           #tonSetStableWeight[#i](IN := #runTaimerStableWeight[#i],
                                   PT := t#250ms);

       ELSE
           #currentWeight[#i] := 0;
           #prevWeight[#i]:= 0;
       END_IF;

       IF #tonSetStableWeight[#i].Q OR #RS_TRIG_openBunker[#i] THEN
           IF #currentWeight[#i] <> "signalKVSStation".stableWeight[#i].weight[0] THEN
               "pushToArray"(addValue := #currentWeight[#i],
                             "array" := #stableWeight[#i].weight);
           END_IF;
           #runTaimerStableWeight[#i] := false;
       END_IF;


   END_FOR;
END_REGION
END_FUNCTION_BLOCK

FUNCTION_BLOCK "Sorting_AM"   // FB13, LAD
TITLE = Блок сортировки
{ S7_Optimized_Access := 'TRUE' }
VERSION : 0.1
// Из массива ReadyToSort считываем количество заполненых бункеров. Если их больше либо равно 6 то начинаем сортировку.
// После нахождения искомых бункеров формируем массив readyToDrop.
// После путем перемножения ReadyToSort *Not(readyToDrop) исключаем сбрасывемые бункера из сортировки
// stored: AutoNumber true, IsIECCheckEnabled false, IsRetainMemResEnabled false, MemoryReserve 100, SetENOAutomatically false, UDAEnableTagReadback false
   VAR_INPUT
      enableToWork : Bool;   // разрешение на работу блока
      setWeight : Real;   // итоговый разыскиваемый вес
      errorMeasurement : Real;   // погрешность
      isWorkWithBunker : Array[0..12] of Bool;   // разрешение работать с конкретными бункерами
      setWeightBunker { ExternalAccessible := 'False'; ExternalVisible := 'False'; ExternalWritable := 'False'} : Array[0..12] of Real;   // уставки весов в бункерах
   END_VAR
   VAR_IN_OUT
      stableWeightBunker : Array[0..12] of Real;   // стабильный вес в бункерах
      readyToSorting : Array[0..12] of Bool;   // готовность бункеров к сортировке
      readyToDrop : Array[0..12] of Bool;   // итоговый сигнал сортировки для сброса на конвейер
      blockSort : Bool;   // блокировать сортировку чтобы просто скинуть все готовые
   END_VAR
   VAR
      valueReadyToDrop { ExternalAccessible := 'False'; ExternalVisible := 'False'; ExternalWritable := 'False'} : Bool;
      valueReadytoSortBunker : SInt;   // количество бункеров готовых к сортировке
      valueIsWorkWithBunker : SInt;
      tmpStableWeight : Array[0..12] of Real;   // массив с весами которые будем сортировать
      bufferReadyToDrop : Array[0..12] of Bool;   // на случай того что если readyToDrop не был сброшен
      Sort_Real_FB : "Sort_Real";
      full1 : Array[0..12] of Bool;
      full0 : Array[0..12] of Bool;
      pow2_DB : "pow2";
      minValue : Real;
      minValueArray : Array[0..12] of Bool;
      tmpArrNotDrop { ExternalAccessible := 'False'; ExternalVisible := 'False'; ExternalWritable := 'False'} : Array[0..12] of Real;
      tmpSumFind { ExternalAccessible := 'False'; ExternalVisible := 'False'; ExternalWritable := 'False'} : Real;
      valueMaxSortFor { ExternalAccessible := 'False'; ExternalVisible := 'False'; ExternalWritable := 'False'} : Int;   // максимальное число циклов для нахождения искомого веса
      bitMaskSortFor { ExternalAccessible := 'False'; ExternalVisible := 'False'; ExternalWritable := 'False'} : Array[0..12] of Bool;
      stateFindIndex { ExternalAccessible := 'False'; ExternalVisible := 'False'; ExternalWritable := 'False'} : Bool;
      tmpReadyToDrop { ExternalAccessible := 'False'; ExternalVisible := 'False'; ExternalWritable := 'False'} : Array[0..12] of Bool;   // временный массив готовности к сбросу
      tabActiveSort { ExternalAccessible := 'False'; ExternalVisible := 'False'; ExternalWritable := 'False'} : Bool;
      saveBitMaskSortFor { ExternalAccessible := 'False'; ExternalVisible := 'False'; ExternalWritable := 'False'} : Array[0..12] of Bool;
   END_VAR
   VAR_TEMP
      i : DInt;
      j : DInt;
      k : DInt;
      l : DInt;
      "m" : DInt;
      it : DInt;
      one : DInt;
      indexTmpSumFind : DInt;
      valueOneBitMask : DInt;
   END_VAR
   // full1[1..12] := true;
BEGIN

REGION Network 1 (SCL): Определяем ValueToSortBunker
   #tmpReadyToDrop := #full0;
   IF #enableToWork THEN //разрешение на работу блока 
       //необходимо проверить не подготовил ли блок сортировки уже значения для сброса
       #valueReadyToDrop := false;
       #i := 0;
       FOR #i := 1 TO 12 DO
           IF #readyToDrop[#i] THEN
               #valueReadyToDrop := true;
               EXIT;//выходим из FOR тк то что надо уже нашли
           END_IF;
       END_FOR;

       IF NOT (#valueReadyToDrop) THEN
           //если сортировку не производили
           #i := 0;
           #valueIsWorkWithBunker := 0;
           #valueReadytoSortBunker := 0;
           FOR #i := 1 TO 12 DO
               //подсчитаем количесво бункеров с которыми можно работать
               //и какие готовы к сортировке
               //
               IF #isWorkWithBunker[#i] THEN
                   #valueIsWorkWithBunker := #valueIsWorkWithBunker + 1;
               END_IF;
               IF #readyToSorting[#i] AND #isWorkWithBunker[#i] THEN
                   #valueReadytoSortBunker := #valueReadytoSortBunker + 1;
               END_IF;
           END_FOR;

           IF #blockSort THEN
               //если включена блокировка то просто ждем готовности бункеров к сортировке
               //
               IF #valueIsWorkWithBunker = #valueReadytoSortBunker THEN
                   //если число готовых к сортировке бункеров совпадает 
                   //с числом разрешенных к работе в режиме блокировки то
                   //просто скидываем все
                   #tmpReadyToDrop := #readyToSorting;
               END_IF;
           ELSE
               //если блокировки нет то сортируем по стандарту

               // IF #valueIsWorkWithBunker = 1 THEN
               //     //если бункеров разрешенных к работе один то 
               //     #i := 0;
               //     FOR #i := 1 TO 12 DO //заполняем временный массив готовности к сбросу
               //         #tmpReadyToDrop[#i] := #readyToSorting[#i] AND #isWorkWithBunker[#i];
               //     END_FOR;
               // ELSE

               //IF #valueReadytoSortBunker >= 3 THEN//начинаем сортировку
               IF #valueReadytoSortBunker =12 THEN//начинаем сортировку
                   #i := 0;
                   FOR #i := 1 TO 12 DO//определим массив чисел с которыми будем работать
                       #tmpStableWeight[#i] := #stableWeightBunker[#i] * BOOL_TO_INT(#readyToSorting[#i]);
                   END_FOR;
                   //далее работаем только с весами из массива #tmpStableWeight
                   //
                   REGION
                       // // //*****************************
                       // // //временная заглушка - скидываем бункера которые тупа в сумме
                       // // //дают больше либо равно уставке
                       // // //
                       // #tmpArrNotDrop := #tmpStableWeight;


                       // //#Sort_Real_FB(array := #tmpArrNotDrop,sortDirection:=true);
                       // //теперь массив #tmpArrNotDrop отсортирован и числа которые 
                       // //мы можем использовать начинаются с индекса (12-noDrop+1)
                       // #k := 0;
                       // #tmpSumFind := 0;//где храним сумму
                       // #stateFindIndex := false;
                       // #indexTmpSumFind := 0;//индекс элемента массива на котором надо остановиться
                       // //#noDrop := #valueReadytoSortBunker;
                       // FOR #k := 0 TO 12 DO
                       //     #tmpSumFind := #tmpSumFind + #tmpArrNotDrop[#k];
                       //     IF #tmpSumFind >= #setWeight//если попадаем 
                       //     THEN
                       //         #stateFindIndex := true;
                       //         #indexTmpSumFind := #k;
                       //         EXIT;//выходим из FOR
                       //     END_IF;

                       // END_FOR;
                       // IF NOT (#stateFindIndex) THEN //ничего не нашли
                       //     #tmpReadyToDrop := #full0;
                       // ELSE
                       //     #l := 0;//заполняем массив на сброс
                       //     FOR #l := 1 TO #indexTmpSumFind DO
                       //         IF #tmpArrNotDrop[#l] > 0 THEN
                       //             #tmpReadyToDrop[#l] := true;
                       //         ELSE
                       //             #tmpReadyToDrop[#l] := false;
                       //         END_IF;
                       //     END_FOR;

                       // END_IF;
                       // // // //*************************************
                   END_REGION ;
                   REGION
                       //****************
                       //сортировка на основе двоичного представления числа
                       //
                       #tmpArrNotDrop := #tmpStableWeight;
                       #Sort_Real_FB("array" := #tmpArrNotDrop,
                                     sortDirection := true);
                       // //теперь массив #tmpArrNotDrop отсортирован в порядке убывания и 
                       //только необходимо обратить внимание что все веса начинаются с 0 индекса
                       #pow2_DB(basic := #valueReadytoSortBunker,
                                pow := #valueMaxSortFor);
                       #it := 0;
                       #stateFindIndex := false;
                       #minValue := 99999;
                       #minValueArray := #full0;
                       #tabActiveSort := false;
                       FOR #it := 1 TO #valueMaxSortFor DO
                           // // #bitMaskSortFor[0] := #it.%X0;
                           // // #bitMaskSortFor[1] := #it.%X1;
                           // // #bitMaskSortFor[2] := #it.%X2;
                           // // #bitMaskSortFor[3] := #it.%X3;
                           // // #bitMaskSortFor[4] := #it.%X4;
                           // // #bitMaskSortFor[5] := #it.%X5;
                           // // #bitMaskSortFor[6] := #it.%X6;
                           // // #bitMaskSortFor[7] := #it.%X7;
                           // // #bitMaskSortFor[8] := #it.%X8;
                           // // #bitMaskSortFor[9] := #it.%X9;
                           // // #bitMaskSortFor[10] := #it.%X10;
                           // // #bitMaskSortFor[11] := #it.%X11;
                           // // #bitMaskSortFor[12] := #it.%X12;
                           // // #tmpSumFind := #tmpArrNotDrop[0] * BOOL_TO_SINT(#bitMaskSortFor[0]) +
                           // // #tmpArrNotDrop[1] * BOOL_TO_SINT(#bitMaskSortFor[1]) +
                           // // #tmpArrNotDrop[2] * BOOL_TO_SINT(#bitMaskSortFor[2]) +
                           // // #tmpArrNotDrop[3] * BOOL_TO_SINT(#bitMaskSortFor[3]) +
                           // // #tmpArrNotDrop[4] * BOOL_TO_SINT(#bitMaskSortFor[4]) +
                           // // #tmpArrNotDrop[5] * BOOL_TO_SINT(#bitMaskSortFor[5]) +
                           // // #tmpArrNotDrop[6] * BOOL_TO_SINT(#bitMaskSortFor[6]) +
                           // // #tmpArrNotDrop[7] * BOOL_TO_SINT(#bitMaskSortFor[7]) +
                           // // #tmpArrNotDrop[8] * BOOL_TO_SINT(#bitMaskSortFor[8]) +
                           // // #tmpArrNotDrop[9] * BOOL_TO_SINT(#bitMaskSortFor[9]) +
                           // // #tmpArrNotDrop[10] * BOOL_TO_SINT(#bitMaskSortFor[10]) +
                           // // #tmpArrNotDrop[11] * BOOL_TO_SINT(#bitMaskSortFor[11]) +
                           // // #tmpArrNotDrop[12] * BOOL_TO_SINT(#bitMaskSortFor[12]);
                           // 
                           #tmpSumFind :=
                           #tmpArrNotDrop[0] * BOOL_TO_SINT(#it.%X0) +
                           #tmpArrNotDrop[1] * BOOL_TO_SINT(#it.%X1) +
                           #tmpArrNotDrop[2] * BOOL_TO_SINT(#it.%X2) +
                           #tmpArrNotDrop[3] * BOOL_TO_SINT(#it.%X3) +
                           #tmpArrNotDrop[4] * BOOL_TO_SINT(#it.%X4) +
                           #tmpArrNotDrop[5] * BOOL_TO_SINT(#it.%X5) +
                           #tmpArrNotDrop[6] * BOOL_TO_SINT(#it.%X6) +
                           #tmpArrNotDrop[7] * BOOL_TO_SINT(#it.%X7) +
                           #tmpArrNotDrop[8] * BOOL_TO_SINT(#it.%X8) +
                           #tmpArrNotDrop[9] * BOOL_TO_SINT(#it.%X9) +
                           #tmpArrNotDrop[10] * BOOL_TO_SINT(#it.%X10) +
                           #tmpArrNotDrop[11] * BOOL_TO_SINT(#it.%X11);

                           IF #tmpSumFind >= #setWeight AND #tmpSumFind <= (#setWeight + (#setWeight * #errorMeasurement / 100))
                           THEN
                               #stateFindIndex := true;
                               EXIT;
                               ;
                           ELSE
                               IF (#tmpSumFind > #setWeight) AND (#tmpSumFind < #minValue) THEN
                                   #minValue := #tmpSumFind;
                                   "bitMaskSortFor"(value := #it,
                                                    bitMask := #bitMaskSortFor);
                                   #minValueArray := #bitMaskSortFor;
                               END_IF;
                           END_IF;


                       END_FOR;
                       //на выходе мы имеем битовую маску которая лучше всего подходит
                       //
                       //также обрабатываем условие что карманы все заняты а чтото скинуть надо
                       IF NOT (#stateFindIndex) THEN //
                           IF #valueReadytoSortBunker > 10 THEN
                               #tabActiveSort := TRUE;
                               #saveBitMaskSortFor := #minValueArray;
                           END_IF;
                       ELSE
                           #tabActiveSort := true;
                           "bitMaskSortFor"(value := #it,
                                            bitMask := #bitMaskSortFor);
                           #saveBitMaskSortFor := #bitMaskSortFor;
                       END_IF;
                       #tmpReadyToDrop := #full0;
                       //определяем финальный tmpReadyToDrop
                       IF #tabActiveSort THEN
                           //если активированная нахождение искомых бункеров
                           #l := 0;
                           FOR #l := 0 TO 12 DO
                               IF #saveBitMaskSortFor[#l] AND ((BOOL_TO_INT(#saveBitMaskSortFor[#l]) * #tmpArrNotDrop[#l]) > 0) THEN
                                   #k := 0;
                                   FOR #k := 1 TO 12 DO
                                       IF #tmpArrNotDrop[#l] = #tmpStableWeight[#k] THEN
                                           #tmpReadyToDrop[#k] := true;
                                           EXIT;
                                       END_IF;
                                   END_FOR;
                               END_IF;
                           END_FOR;
                       END_IF;
                   END_REGION
                   //корректируем массив readyToSorting
                   #i := 0;
                   FOR #i := 1 TO 12 DO
                       IF #tmpReadyToDrop[#i] THEN
                           #readyToSorting[#i] := false;
                       END_IF;
                   END_FOR;
               END_IF;
           END_IF;
       ELSE
           #tmpReadyToDrop := #readyToDrop;//если значения уже были
           //и не сброшены то сортировку не производили
       END_IF;

   END_IF;



   #readyToDrop := #tmpReadyToDrop;//переписываем из временного в блочный
END_REGION
END_FUNCTION_BLOCK

FUNCTION_BLOCK "pow2"
{ S7_Optimized_Access := 'TRUE' }
VERSION : 0.1
   VAR_INPUT 
      basic : SInt;   // степень возведение двойки
   END_VAR

   VAR_IN_OUT 
      pow : Int;   // ответ возведения -1
   END_VAR


BEGIN
	CASE #basic OF //
	    1:
	       #pow:=1;
	    2:  
	        #pow:=3;
	    3:
	        #pow:=7;
	    4:
	        #pow:=15;
	    5:
	        #pow:=31;
	    6:
	        #pow:=63;
	    7:
	        #pow:=127;
	    8:
	        #pow:=255;
	    9:
	        #pow:=511;
	    10:
	        #pow:=1023;
	    11:
	        #pow:=2047;
	    12:
	        #pow:=4095;
	END_CASE;
	
END_FUNCTION_BLOCK

FUNCTION_BLOCK "setWeightBunker_AM"   // FB3, LAD
{ S7_Optimized_Access := 'TRUE' }
VERSION : 0.1
// Блок уставок, работы упаковочных машин.
// Определяет уставки для бункеров. Дают разрешение на работу бункера.
// Даже если сброшено меньше 
// Говорит о готовности упаковочных машин принять дозу и в какую машину скидывать
// stored: AutoNumber true, IsIECCheckEnabled false, IsRetainMemResEnabled false, MemoryReserve 100, SetENOAutomatically false, UDAEnableTagReadback false
   VAR_INPUT
      enableWork : Bool;   // разрешение работы блока
      weightPack : Real;   // заданный вес упаковки
      measurementError : Real;   // погрешность
      maxWeightBunker : Real;   // максимальный вес в бункере
      mediumWeightProduct : Real;   // средний вес продукта
   END_VAR
   VAR_IN_OUT
      taskWeightBunker : Real;   // целевой вес который ищем в сортировке
      setWeightBunker : Array[0..12] of Real;   // уставки задаваемые в бункера
      isWorkWithBunker : Array[0..12] of Bool;   // разрешение работать с конкретными бункерами
      readyToDrop : Array[0..12] of Bool;   // массив который будет сбрасываться
      YP_ReadyToDrop : Array[0..2] of Bool;   // сигнал говорит о том что в УМ можно 100% чтото скинуть
      stableWeightBunker : Array[0..12] of Real;   // стабильный вес в бункерах
      blockSort : Bool;   // запрещение работы сортировки в блоке сортировки
   END_VAR
   VAR
      measureErrorGramm : Real;   // погрешность измерения в граммах
      dropWeight : Real;   // уже сброшенный вес
      hmiDropWeight : Real;   // отображаемый сброшенный вес на панеле
      hmiMeasurementError : Real;   // отображаемая сброшенная погрешность на панеле
      indexLastDropYP : SInt;   // индекс машины в которую последний раз сбрасывали
      full1 : Array[0..12] of Bool;
      full0 : Array[0..12] of Bool;
      Sort_Real_FB : "Sort_Real";
   END_VAR
   VAR_TEMP
      i : DInt;
      j : DInt;
      k : DInt;
      l : DInt;
      "m" : DInt;
      expX : Real;
      expY : Real;
      tmpNeedWeight : Real;
      tmpc1 : Real;
      tmpc2 : DInt;
      tmpc3 : Real;
      minSearch : Real;   // минимальное найденое число остаточном массиве
      indexMinSearch : DInt;   // индекс минимального числа
      isSearchSuccess : Bool;   // поиск прошел успешно
      indexSearchSuccess : DInt;   // индекс оставшегося идеального кармана
      valueDropBunker : DInt;
      tmpArrNotDrop : Array[0..12] of Real;
      tmpArrWeightNoDrop : Array[0..12] of Real;
      noDrop : Int;
      tmpSumFind : Real;
      indexTmpSumFind : DInt;
   END_VAR
   // full1[1..12] := true;
BEGIN

REGION Network 1 (SCL): переведем погрешность в граммы
   #measureErrorGramm := #measurementError * #weightPack / 100;
END_REGION

REGION Network 2 (SCL): Определяем уставки в карманы и выставляем разрешения работы
   // на основе веса который мы уже сбросили и который будем сбрасывать 
   // а также учитывая веса в рецепте определяем уставки в карманах, целевую уставку для поиска, а также 
   // выставляем разрешения работы по конкретным бункерам
   IF #enableWork THEN

       //*********************************************
       //определение сброшенного веса на основе массивов со стабильными весами
       //и массива ячеек которые должны быть сброшены. Обнуление сброшенного веса в случае 
       //выполнения условия
       //также производим этот расчет только при условии что мы сбросим кудато этот вес
       IF #YP_ReadyToDrop[1] OR #YP_ReadyToDrop[2] THEN
           #i := 0;
           FOR #i := 1 TO 12 DO
               #dropWeight := #dropWeight + BOOL_TO_INT(#readyToDrop[#i]) * #stableWeightBunker[#i];
           END_FOR;
           // #hmiDropWeight := #dropWeight;
           // #hmiMeasurementError := (#weightPack - #dropWeight) / #weightPack;
           IF #dropWeight >= #weightPack THEN
               #dropWeight := 0;
           END_IF;
       END_IF;
       //************************************


       //основное распространение весов, когда выкидываем весь вес за раз
       //

       #expX := #weightPack / 10;//#weightPack / 6;
       #expY := #mediumWeightProduct / 3;

       //если #expX<=MAX_WEIGHT_BUNKER то работаем по стандарту,
       //иначе ограничеваем #expX=MAX_WEIGHT_BUNKER
       IF #expX > #maxWeightBunker THEN
           #expX := #maxWeightBunker;
       END_IF;

       IF #dropWeight = 0 THEN
           // #j := 2;
           // WHILE (6 * #expX) < #weightPack + #j * #expY AND #j <> 0 DO
           //     #j := #j - 1;
           // END_WHILE;
           // #expY := (#expY / 2) * #j;//корректировка #expY
           #taskWeightBunker := #weightPack;//вес для поиска по рецепту
           #isWorkWithBunker := #full1;//разрешаем работу всем линиям

           #setWeightBunker[1] := #setWeightBunker[6] :=
           #setWeightBunker[7] := #setWeightBunker[12] := #expX;

           #setWeightBunker[2] := #setWeightBunker[5] :=
           #setWeightBunker[8] := #setWeightBunker[11] := #expX - #expY;

           #setWeightBunker[3] := #setWeightBunker[4] :=
           #setWeightBunker[9] := #setWeightBunker[10] := #expX - 2 * #expY;

       ELSE//если уже сбрасываем

           #valueDropBunker := 0;//определяем сбрасываем ли мы чтото чтобы запретить
           //перерасчет в этом условии
           //просто на первой итерации как только сюда поступает массив readyToDrop
           //мы выставляем требуемые уставки, а потом запрещаем их изменять
           #k := 0;
           FOR #k := 1 TO 12 DO
               #valueDropBunker := #valueDropBunker + BOOL_TO_SINT(#readyToDrop[#k]);
           END_FOR;

           IF #valueDropBunker > 0 THEN
               //следующий просчет актуален только на итерации перед сбросом веса поэтому 
               //после сброса на конвейер эту часть надо блокировать для изменений
               //
               //только еще надо обыгрывать момент когда сбрасываются сразу 12 бункеров

               #tmpNeedWeight := #weightPack - #dropWeight;//вес остатка

               IF #valueDropBunker < 12 THEN //при сбрасывании всех 12 бункеров
                   //будет другой механизм выдачи разрешений

                   IF #tmpNeedWeight <= #expX THEN //если нужно докинуть меньше чем в одном бункере,то
                       //ищем вес совпадающий с остатком и если такой не находим
                       //то берем минимальную ячейку с весом

                       #minSearch := 99999.9;//берется как минимальное тк такое точно не будет в бункере
                       #k := 0;
                       #isSearchSuccess := false;
                       FOR #k := 1 TO 12 DO//ищем бункер идеально подходящий по весу и параллельно ведем
                           //поиск первого минимального числа

                           IF NOT (#readyToDrop[#k]) THEN
                               IF #stableWeightBunker[#k] < #minSearch THEN
                                   //параллельно ищем минимальное число
                                   #minSearch := #stableWeightBunker[#k];
                                   #indexMinSearch := #k;
                               END_IF;

                               IF (#tmpNeedWeight <= #stableWeightBunker[#k]//проверяем оставшиеся карманы на вес
                                   AND #stableWeightBunker[#k] <= #tmpNeedWeight + #measureErrorGramm / 6) THEN
                                   #isSearchSuccess := true;
                                   #indexSearchSuccess := #k;//сохраняем индекс идеального кармана
                                   EXIT;//выходим из FOR
                               END_IF;
                           END_IF;

                       END_FOR;
                       //если идеальный карман так и не найдем 
                       //берем карман с минимальным весом и перемещаем его индекс в #indexSearchSuccess
                       IF NOT (#isSearchSuccess) THEN
                           #indexSearchSuccess := #indexMinSearch;
                       END_IF;

                       #taskWeightBunker := #tmpNeedWeight;//вес для поиска в сортировке
                       #isWorkWithBunker := #full0;//запрещаем работу всем линиям
                       #isWorkWithBunker[#indexSearchSuccess] := true;//включаем только нужную линию
                       #setWeightBunker[#indexSearchSuccess] := #tmpNeedWeight;
                       #blockSort := true;//выставляем блокировку тк надо будет только сбросить

                   ELSE//если докидывать больше чем в одном бункере
                       #k := 0;//выделяем веса которые не сбрасываются
                       FOR #k := 1 TO 12 DO
                           IF NOT (#readyToDrop[#k]) THEN
                               #noDrop := #noDrop + 1;//колво добавленных элементов
                               #tmpArrNotDrop[#k] := #stableWeightBunker[#k];
                           END_IF;
                       END_FOR;
                       //будем использовать #tmpArrWeightNoDrop для поиска искомых бункеров
                       #tmpArrWeightNoDrop := #tmpArrNotDrop;

                       #Sort_Real_FB("array" := #tmpArrNotDrop);
                       //теперь массив #tmpArrNotDrop отсортирован и числа которые 
                       //мы можем использовать начинаются с индекса (12-noDrop+1)
                       #k := 0;
                       #tmpSumFind := 0;//где храним сумму
                       #indexTmpSumFind := 0;//индекс элемента массива на котором надо остановиться
                       FOR #k := (12 - #noDrop + 1) TO 12 DO
                           #tmpSumFind := #tmpSumFind + #tmpArrNotDrop[#k];
                           IF #tmpSumFind >= #tmpNeedWeight//если попадаем идеально
                               AND #tmpSumFind <= #tmpNeedWeight + #measureErrorGramm THEN
                               #indexTmpSumFind := #k;
                               EXIT;//выходим из FOR
                           END_IF;
                           //если превысили сумму
                           IF #tmpSumFind > #tmpNeedWeight + #measureErrorGramm THEN
                               #indexTmpSumFind := #k - 1;
                               EXIT;
                           END_IF;
                           IF #k = 12 THEN
                               #indexTmpSumFind := #k;
                           END_IF;
                       END_FOR;
                       //теперь проверим чтобы #indexTmpSumFind входил в массив с весами
                       //потому что первый же вес может быть больше того что мы исчем
                       IF #tmpArrNotDrop[#indexTmpSumFind] <> 0 THEN
                           #taskWeightBunker := #tmpNeedWeight;//вес для поиска по рецепту
                           #isWorkWithBunker := #full0;//запрещаем работу всем линиям
                           #blockSort := true;//выставляем блокировку тк надо будет только
                           //дождать сигналов готовности к сортировке сбросить

                           //теперь заполняем массив разрешения работ через поиск весов
                           //и параллельно выставляем уставки
                           IF #tmpSumFind >= #tmpNeedWeight//если попадаем идеально
                               AND #tmpSumFind <= #tmpNeedWeight + #measureErrorGramm THEN
                               //если вес сходился 
                               #l := 0;
                               FOR #l := (12 - #noDrop + 1) TO #indexTmpSumFind DO
                                   #m := 0;
                                   FOR #m := 1 TO 12 DO//ищем отсортированные веса и сопоставляем их индексы
                                       //ищем в заранее сохранненом массивве с весам который не сбрасываются
                                       //и имеют правильные индексы
                                       IF #tmpArrWeightNoDrop[#m] = #tmpArrNotDrop[#l] THEN
                                           #isWorkWithBunker[#m] := true;
                                           #setWeightBunker[#m] := #tmpArrWeightNoDrop[#m];
                                           EXIT;//ищем следующий вес
                                       END_IF;
                                   END_FOR;
                               END_FOR;

                           ELSE //сюда поподем если веса с излишкой или недостаточно 
                               //если вес не сходился
                               #l := 0;
                               FOR #l := (12 - #noDrop + 1) TO #indexTmpSumFind DO
                                   #m := 0;
                                   FOR #m := 1 TO 12 DO
                                       IF #tmpArrWeightNoDrop[#m] = #tmpArrNotDrop[#l] THEN
                                           #isWorkWithBunker[#m] := true;
                                           #setWeightBunker[#m] := #tmpNeedWeight / DINT_TO_INT((#indexTmpSumFind - (12 - #noDrop + 1)));
                                           EXIT;//ищем следующий вес
                                       END_IF;
                                   END_FOR;
                               END_FOR;


                           END_IF;
                           ;

                       END_IF;

                   END_IF;
               ELSE //а теперь что делать если сброшены все 12
                   //надо вводить какойто новый сигнал который сказал бы нагружать бункера только после закрытия? или 
                   //все успеется
                   //!!!обратить внимание на это
                   //

                   //расчитываем сколько бункеров необходимо для сбора оставшегося веса
                   //это делаем на основе максимального веса в бункере
                   //
                   #taskWeightBunker := #tmpNeedWeight;//вес для поиска в сортировке
                   #blockSort := true;//выставляем блокировку тк надо будет только скинуть
                   #tmpc2 := ROUND(#tmpNeedWeight / #maxWeightBunker); //число используемых бункеров
                   #i := 0;
                   FOR #i := 1 TO #tmpc2 DO
                       #isWorkWithBunker[#k] := true;
                       #setWeightBunker[#k] := #tmpNeedWeight / DINT_TO_REAL(#tmpc2);
                   END_FOR;
                   ;
               END_IF;
           END_IF;
       END_IF;


   ELSE
       #isWorkWithBunker := #full0;//запрет на работу все бункерам
   END_IF;
END_REGION
END_FUNCTION_BLOCK

FUNCTION_BLOCK "workPackingMachine_AM"   // FB4, LAD
TITLE = Работа с УМ, бункерами
{ S7_Optimized_Access := 'TRUE' }
VERSION : 0.1
// stored: AutoNumber true, IsIECCheckEnabled false, IsRetainMemResEnabled false, MemoryReserve 100, SetENOAutomatically false, UDAEnableTagReadback false
   VAR_INPUT
      enWork : Bool;   // разрешение работы
      YP_ReadyAccept : Array[0..2] of Bool;   // сигнал от упак машины что готова принять
      YP_StartDozing : Array[0..2] of Bool;   // сигнал от упаковочной машины что начать дозирование
      weightPack : Real;   // заданный вес упаковки
   END_VAR
   VAR_IN_OUT
      hmiYpDropWeight : Array[0..2] of Real;   // вывод на панель сброшенного веса
      hmiYPDropErrorMeasure : Array[0..2] of Real;   // вывод на панель погрешности
      openLeftBunker : Array[0..12] of Bool;   // сгналы открытия левых бункеров
      closeLeftBunker : Array[0..12] of Bool;   // сигналы закрытия левых бункеров
      openRightBunker : Array[0..12] of Bool;   // сигналы открытия правых бункеров
      closeRightBunker : Array[0..12] of Bool;   // сигналы закрытия правых бункеров
      alarmStop : Bool;   // аварийный останов
      Yq_ReadyDoze : Array[0..2] of Bool;   // сигнал на упаковочную машину что доза готова
      YP_ReadyToDrop : Array[0..2] of Bool;   // сигнал говорит о том что в УМ можно 100% чтото скинуть
      stableWeightBunker : Array[0..12] of Real;   // стабильный вес в бункерах
      readyToSort : Array[0..12] of Bool;
      readyToDrop : Array[0..12] of Bool;   // массив который будет сбрасываться
      Conv_FRV : Array[0..2] of Bool;   // запуск конвейеров вперед
      Conv_REV : Array[0..2] of Bool;   // запуск конвейеров назад
   END_VAR
   VAR
      dropLeftBunker { ExternalAccessible := 'False'; ExternalVisible := 'False'; ExternalWritable := 'False'} : Array[0..12] of Bool;   // массив на сброс левых бункеров
      dropRightBunker { ExternalAccessible := 'False'; ExternalVisible := 'False'; ExternalWritable := 'False'} : Array[0..12] of Bool;   // массив на сброс правых бункеров
      tmpPtrig : Array[0..1] of Bool;
      dropTon : Array[0..2] of TON_TIME;   // выдержка на передачу сигнала УМ ДОЗА
      startDropTon : Array[0..2] of Bool;   // начало отсчета для таймера
      dropWeight : Real;   // сбрасываемый вес
      nextDropConveyer : SInt;   // индекс конвейера на который сбрасывали последним
      tonReadyDozeTimer : Array[0..2] of TON_TIME;
      leftBunker_FB : Array[0..12] of "controlValve";
      rightBunker_FB : Array[0..12] of "controlValve";
      full1 : Array[0..12] of Bool;
      full0 : Array[0..12] of Bool;
      valueDropBunker : Bool;
      watchDrop : Array[0..12] of Bool;
      F_TRIG_Instance { S7_SetPoint := 'True'} : F_TRIG;
   END_VAR
   VAR_TEMP
      i : DInt;
      resetTimerDropYp : Array[0..2] of Bool;
      resetTimerDropTon : Array[0..2] of Bool;
   END_VAR
   // full1[1..12] := true;
   VAR_TEMP   // added for the SCL form of the ladder/FBD networks
      _w1 : Bool;
      _w2 : Bool;
   END_VAR
BEGIN

REGION Network 1: сброс вращения если убрать сигнал разрешения
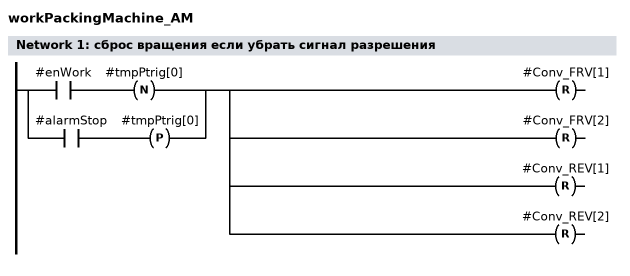
   RUNG wire#powerrail
      Contact( #enWork )
      N_Trig( #tmpPtrig[0] )
      wire#w1
      R_Coil( #Conv_FRV[1] )
   END_RUNG
   RUNG wire#powerrail
      Contact( #alarmStop )
      P_Trig( #tmpPtrig[0] )
   END_RUNG wire#w1
   RUNG wire#w1
      R_Coil( #Conv_FRV[2] )
   END_RUNG
   RUNG wire#w1
      R_Coil( #Conv_REV[1] )
   END_RUNG
   RUNG wire#w1
      R_Coil( #Conv_REV[2] )
   END_RUNG
   // the same network as SCL:
   #_w1 := NOT #enWork AND #tmpPtrig[0];   // falling edge
   #tmpPtrig[0] := #enWork;
   #_w2 := #alarmStop AND NOT #tmpPtrig[0];   // rising edge
   #tmpPtrig[0] := #alarmStop;
   IF #_w1 OR #_w2 THEN
       #Conv_FRV[1] := FALSE;
       #Conv_FRV[2] := FALSE;
       #Conv_REV[1] := FALSE;
       #Conv_REV[2] := FALSE;
   END_IF;
END_REGION

REGION Network 2 (SCL): Подсчет сбрасываемых бункеров
   #i := 0;
   #valueDropBunker := FALSE;
   FOR #i := 1 TO 12 DO
       IF #readyToDrop[#i] THEN
           #valueDropBunker := true;
           EXIT;
       END_IF;
   END_FOR;
END_REGION

REGION Network 3 (SCL): Сброс сигнала на УМ #Yq_ReadyDoze
   #i := 0;
   FOR #i := 1 TO 2 DO
       // IF #Yq_ReadyDoze[#i] THEN
       //     #Yq_ReadyDoze[#i] := false;
       // END_IF;
       #tonReadyDozeTimer[#i](IN := #Yq_ReadyDoze[#i],
                              PT := t#1s,
                              Q => #resetTimerDropYp[#i]);

   END_FOR;
   #i := 0;
   FOR #i := 1 TO 2 DO

       IF #resetTimerDropYp[#i] THEN
           #Yq_ReadyDoze[#i] := false;
       END_IF;

   END_FOR;
END_REGION

REGION Network 4 (SCL): Формирование сигналов
   // #YP_ReadyToDrop
   #i := 0;
   FOR #i := 1 TO 2 DO
       #YP_ReadyToDrop[#i] := #YP_ReadyAccept[#i] AND #YP_StartDozing[#i] AND NOT(#startDropTon[#i]) AND NOT(#Yq_ReadyDoze[#i]);
   END_FOR;
END_REGION

REGION Network 5 (SCL): учет сбрасываемого веса
   // помещаем в переменнную #dropWeight вес который будет сброшен
   IF #enWork THEN
       IF (#YP_ReadyToDrop[1] OR #YP_ReadyToDrop[2]) AND #valueDropBunker THEN
           #i := 0;
           FOR #i := 1 TO 12 DO
               #dropWeight := #dropWeight + BOOL_TO_INT(#readyToDrop[#i])
               * #stableWeightBunker[#i];
           END_FOR;
       END_IF;
   END_IF;
END_REGION

REGION Network 6 (SCL): вращение конвейеров
   //"hmi".outConvAndPack[1].isUseInBegin - разрешение использовать
   // "hmi".outConvAndPack[1].isUpInBegin - вращать вперед
   #i := 0;
   FOR #i := 1 TO 2 DO
       IF #enWork AND "hmi".outConvAndPack[#i].isUseInBegin THEN
           IF "hmi".outConvAndPack[#i].isUpInBegin THEN
               #Conv_FRV[#i] := true;
               #Conv_REV[#i] := false;
           ELSE
               #Conv_FRV[#i] := false;
               #Conv_REV[#i] := true;
           END_IF;
       ELSE
           #Conv_FRV[#i] := false;
           #Conv_REV[#i] := false;
       END_IF;
   END_FOR;
END_REGION

REGION Network 7 (SCL): Формирование сигнала доза готова
   IF #enWork THEN
       IF #valueDropBunker THEN//определяем какие бункеры открываем
           //, а также даем отсечку времени для отправки
           //ДОЗА ГОТОВА
           IF #YP_ReadyToDrop[1] OR #YP_ReadyToDrop[2] THEN
               //ПРОСТО ЕСЛИ НЕ СКИДЫВАЕМ ТО И НЕ НАДО ОЧИЩАТЬ МАССИВ READYTOdROP
               IF #YP_ReadyToDrop[1] AND #YP_ReadyToDrop[2] THEN
                   //если оба доступны то по следующему индексу
                   CASE #nextDropConveyer OF
                       0, 2:  //следующий был второй
                           IF #Conv_FRV[2] THEN
                               #hmiYpDropWeight[1] := #dropWeight;
                               #hmiYPDropErrorMeasure[1] := (#weightPack - #dropWeight) / #weightPack * 100;
                               #startDropTon[1] := true;
                           ELSE
                               #hmiYpDropWeight[2] := #dropWeight;
                               #hmiYPDropErrorMeasure[2] := (#weightPack - #dropWeight) / #weightPack * 100;
                               #startDropTon[2] := true;
                           END_IF;
                           #dropLeftBunker := #readyToDrop;

                       1:  // следующий первый
                           IF #Conv_FRV[1] THEN
                               #hmiYpDropWeight[1] := #dropWeight;
                               #hmiYPDropErrorMeasure[1] := (#weightPack - #dropWeight) / #weightPack * 100;
                               #startDropTon[1] := true;
                           ELSE
                               #hmiYpDropWeight[2] := #dropWeight;
                               #hmiYPDropErrorMeasure[2] := (#weightPack - #dropWeight) / #weightPack * 100;
                               #startDropTon[2] := true;
                           END_IF;
                           #dropRightBunker := #readyToDrop;

                   END_CASE;

               ELSE
                   #i := 0;
                   FOR #i := 1 TO 2 DO
                       IF #YP_ReadyToDrop[#i] THEN
                           #hmiYpDropWeight[#i] := #dropWeight;
                           #hmiYPDropErrorMeasure[#i] := (#weightPack - #dropWeight) / #weightPack * 100;
                           #startDropTon[#i] := TRUE;

                           IF (#Conv_FRV[1] AND #Conv_FRV[2]) OR //если конвейера вращаются в одну сторону
                               (#Conv_REV[1] AND #Conv_REV[2]) THEN
                               #dropLeftBunker := #readyToDrop;
                               #dropRightBunker := #readyToDrop;
                               #watchDrop := #readyToDrop;
                           ELSE
                               IF #i = 1 THEN//Если готова только первая УМ
                                   IF #Conv_FRV[1] THEN
                                       #dropRightBunker := #readyToDrop;
                                   ELSE
                                       #dropLeftBunker := #readyToDrop;
                                   END_IF;
                               ELSE//если готова только вторая УМ
                                   IF #Conv_REV[1] THEN
                                       #dropRightBunker := #readyToDrop;
                                   ELSE
                                       #dropLeftBunker := #readyToDrop;
                                   END_IF;

                               END_IF;

                           END_IF;
                           EXIT;//выйти из for если нашли нужную УМ
                       END_IF;
                   END_FOR;
               END_IF;
               #readyToDrop := #full0;
           END_IF;
       END_IF;
   END_IF;

   //изменяем конвейер на который будем скидывать
   IF #dropWeight >= #weightPack AND (#YP_ReadyToDrop[1] OR #YP_ReadyToDrop[2]) THEN
       #dropWeight := 0;
       IF #nextDropConveyer = 0 OR #nextDropConveyer = 2 THEN
           #nextDropConveyer := 1;
       ELSE
           #nextDropConveyer := 2;
       END_IF;
   END_IF;
END_REGION

REGION Network 8 (SCL): открывание левых и правых бункеров
   IF #enWork THEN
       #i := 0;
       FOR #i := 1 TO 12 DO

           #leftBunker_FB[#i](autoclose_M := TRUE,
                              time_autoclose := T#500ms,
                              "time_open/close" := T#200ms,
                              openQ => #openLeftBunker[#i],
                              closeQ => #closeLeftBunker[#i],
                              open := #dropLeftBunker[#i],
                              stopAlarm := #alarmStop);
           #dropLeftBunker[#i] := false;


           #rightBunker_FB[#i](autoclose_M := TRUE,
                               time_autoclose := T#500ms,
                               "time_open/close" := T#200ms,
                               openQ => #openRightBunker[#i],
                               closeQ => #closeRightBunker[#i],
                               open := #dropRightBunker[#i],
                               stopAlarm := #alarmStop);
           #dropRightBunker[#i] := false;

       END_FOR;
   END_IF;

   #F_TRIG_Instance(CLK := #enWork);

   IF #F_TRIG_Instance.Q THEN
       #i := 0;
       FOR #i := 1 TO 12 DO
           #openRightBunker[#i] := false;
           #closeRightBunker[#i] := false;
           #openLeftBunker[#i] := false;
           #closeLeftBunker[#i] := false;
       END_FOR;
   END_IF;
END_REGION

REGION Network 9 (SCL): Формирование сигнала ДОЗА на упаковочную машину
   #i := 0;
   FOR #i := 1 TO 2 DO
       #dropTon[#i](IN := #startDropTon[#i],
                    PT := t#1500ms,
                    Q => #resetTimerDropTon[#i]);

       IF #resetTimerDropTon[#i] THEN
           #Yq_ReadyDoze[#i] := true;
           #startDropTon[#i] := false;
       END_IF;

       "hmi".outConvAndPack[#i].isReadyDozaPackingMachine := #Yq_ReadyDoze[#i];
   END_FOR;
END_REGION
END_FUNCTION_BLOCK

FUNCTION_BLOCK "workInConveyer_AM"   // FB6, LAD
{ S7_Optimized_Access := 'TRUE' }
VERSION : 0.1
// stored: AutoNumber true, IsIECCheckEnabled false, IsRetainMemResEnabled false, MemoryReserve 100, SetENOAutomatically false, UDAEnableTagReadback false
   VAR_INPUT
      enableWork : Bool;   // разрешение работы
      "setSpeed%Int" : Int;   // уставка скорости
      sensorOverflow : Bool;   // датчик пересыпа
   END_VAR
   VAR_OUTPUT
      startinConveyor : Bool;   // запуск конвейера
      "setSpeed%Real" : Real;
   END_VAR
   VAR
      tonOverflowTable : TON_TIME;   // задержка на включение сигнала пересыпа
      tofOverflowTable : TOF_TIME;   // задержка на выключение сигнала пересыпа
      isOverFlowTable : Bool;   // сигнал сработки сигнала пересыпа
   END_VAR
BEGIN

REGION Network 1: сигнал сработки сигнала пересыпа
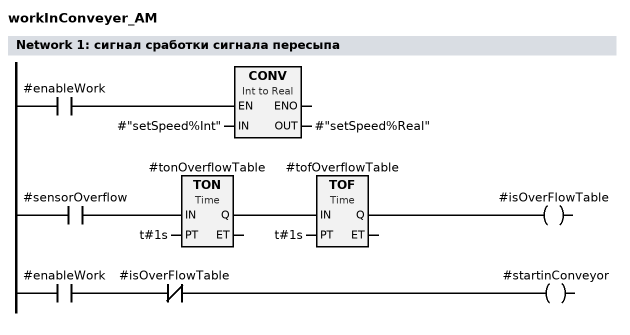
   RUNG wire#powerrail
      Contact( #enableWork )
      { S7_Templates := "[SrcType := Int, DestType := Real]" } Convert(in := #"setSpeed%Int", out => #"setSpeed%Real")
   END_RUNG
   RUNG wire#powerrail
      Contact( #sensorOverflow )
      { S7_Templates := "time_type := Time" } #tonOverflowTable.TON(pt := t#1s, et =>)
      { S7_Templates := "time_type := Time" } #tofOverflowTable.TOF(pt := t#1s, et =>)
      Coil( #isOverFlowTable )
   END_RUNG
   RUNG wire#powerrail
      Contact( #enableWork )
      I_Contact( #isOverFlowTable )
      Coil( #startinConveyor )
   END_RUNG
   // the same network as SCL:
   IF #enableWork THEN #"setSpeed%Real" := INT_TO_REAL(#"setSpeed%Int"); END_IF;
   #tonOverflowTable(IN := #sensorOverflow, PT := t#1s);   // TON
   #tofOverflowTable(IN := #tonOverflowTable.Q, PT := t#1s);   // TOF
   #isOverFlowTable := #tofOverflowTable.Q;
   #startinConveyor := #enableWork AND NOT #isOverFlowTable;
END_REGION
END_FUNCTION_BLOCK

FUNCTION_BLOCK "workVibroLot_AM"   // FB8, LAD
TITLE = Управление линиями вибролотков и вибраций
{ S7_Optimized_Access := 'TRUE' }
VERSION : 0.1
// Если собрано разрешение на работу и ReadyToSort=0 и если вес меньше заданного то включен вибролоток и открыта лопатка
// stored: AutoNumber true, IsIECCheckEnabled false, IsRetainMemResEnabled false, MemoryReserve 100, SetENOAutomatically false, UDAEnableTagReadback false
   VAR_INPUT
      enableWork : Bool;   // разрешение работы
      setWeightBunker : Real;   // уставка веса для бункера
      currentWeight : Real;   // текущий вес
      stateDoor : Bool;   // состояние лопатки
      stateBunkerLeft : Bool;   // состояние левого бункера
      stateBunkerRight : Bool;   // состояние правого бункера
      isWorkWithBunker : Bool;   // разрешение работать с конкретными бункерами
   END_VAR
   VAR_IN_OUT
      onVibroLot : Bool;   // сигнал на включение вибролотков
      closeDoor : Bool;   // сигнал на закрытие лопатки
      openDoor : Bool;   // сигнал на открытие лопатки
      alarmStop : Bool;   // аварийный останов
      isReadyToSort : Bool;   // бункер готов к сортировке
      isReadyToDrop : Bool;   // бункер готов к сбросу
   END_VAR
   VAR
      controlDoor : "controlValve";
      enableWorkAfterCloseDoor : Bool;   // разрешение работы после закрытия бункеров
      tonAfterCloseDoor : TON_TIME;   // выдержка времени после закрытия бункеров
      stateBothBunker : Bool;   // состояние обоих бункеров
      tonToSetSort : TON_TIME;   // выдержка на выставление готов к сортировке
      startToToSetSort : Bool;   // бит на старт таймера выше
      isSetSort : Bool;   // сигнал что бункер готов к сортировке
   END_VAR
   VAR_TEMP
      tmpOpen : Bool;
      tmpClose : Bool;
   END_VAR
BEGIN

REGION Network 1 (SCL): состояние обоих бункеров
   //определим состояние бункеров
   #stateBothBunker := NOT (#stateBunkerLeft) AND NOT (#stateBunkerRight);

   //сигнал выдержки на разрешение работы лотка
   #tonAfterCloseDoor(IN:=#stateBothBunker,
                      PT:=t#300ms,
                      Q=>#enableWorkAfterCloseDoor);
   //сигнал выдержки для выставления состояния готов к сортировке
   #tonToSetSort(IN := #startToToSetSort,
                 PT := t#10ms,
                 Q => #isSetSort);

   IF #isSetSort THEN
       #isReadyToSort := true;
       #startToToSetSort := false;
   END_IF;

   IF #enableWork AND NOT(#alarmStop) THEN//проверяем глобальное разрешение на работу
       IF #currentWeight < #setWeightBunker THEN
           #isReadyToSort := false;
       END_IF;
       IF  #currentWeight<#setWeightBunker AND NOT(#isReadyToSort)
           AND NOT(#isReadyToDrop) AND #isWorkWithBunker
           AND #enableWorkAfterCloseDoor
       THEN
           #startToToSetSort := FALSE;
           #onVibroLot := true;
           IF NOT (#stateDoor) THEN
               #tmpOpen := true;
           END_IF;

       ELSE
           //если мы зашли сюда потому что набрали вес, то заупускаем таймер
           IF #currentWeight >= #setWeightBunker AND NOT(#isReadyToDrop)
               AND NOT(#isReadyToSort) AND #enableWorkAfterCloseDoor THEN
               #startToToSetSort := true;
               // #isSetSort := true;
           END_IF;
           //если зашли сюда потому что уже таймер вышел либо, готовы к сбросу,
           //либо нет разрешений то просто держим лоток выключенным и закрытым
           IF #isReadyToDrop OR #isReadyToSort
               OR NOT(#enableWorkAfterCloseDoor) OR NOT(#isWorkWithBunker)  THEN
               #onVibroLot := false;
               IF #stateDoor THEN
                   #tmpClose := true;
               END_IF;
           END_IF;


       END_IF;

   ELSE
       #isSetSort := false;
       #startToToSetSort := false;
       #isReadyToSort := FALSE;
       #onVibroLot := FALSE;
       #openDoor := FALSE;
       #closeDoor := false;
   END_IF;





   //управление лопаткой
   #controlDoor("time_open/close" := T#250ms,
                openQ => #openDoor,
                closeQ => #closeDoor,
                open := #tmpOpen,
                close := #tmpClose,
                stopAlarm := #alarmStop);
END_REGION
END_FUNCTION_BLOCK

FUNCTION_BLOCK "workVibroTable_AM"   // FB7, LAD
TITLE = Управление вибростолами
{ S7_Optimized_Access := 'TRUE' }
VERSION : 0.1
// На основе массивов готовности бункеров к сортировке решаем работать столу или нет
// stored: AutoNumber true, IsIECCheckEnabled false, IsRetainMemResEnabled false, MemoryReserve 100, SetENOAutomatically false, UDAEnableTagReadback false
   VAR_INPUT
      enableWork : Bool;
      alarmStop : Bool;
      arrayReadyWeightBunker : Array[0..12] of Bool;
   END_VAR
   VAR_OUTPUT
      vibroTable : Array[0..2] of Bool;
   END_VAR
   VAR
      tmpValueReadyWeight : Array[0..2] of Bool;
   END_VAR
   VAR_TEMP
      i : DInt;
   END_VAR
BEGIN

REGION Network 1 (SCL)
   //в массиве arrayReadyWeightBunker храняться состояния готовности веса в бункерах

   IF #enableWork AND NOT(#alarmStop) THEN
       // #tmpValueReadyWeight[1] := true;
       // #tmpValueReadyWeight[2] := true;
       // #i := 0;
       // FOR #i := 1 TO 6 DO
       //     #tmpValueReadyWeight[1] := #tmpValueReadyWeight[1] AND #arrayReadyWeightBunker[#i];
       //     #tmpValueReadyWeight[2] := #tmpValueReadyWeight[2] AND #arrayReadyWeightBunker[#i + 6];
       // END_FOR;
       #i := 0;
       FOR #i := 1 TO 2 DO
           // IF NOT (#tmpValueReadyWeight[#i]) THEN //#tmpValueReadyWeight=0 если хотябы один бункер не готов
               #vibroTable[#i] := true;
           // ELSE
               // #vibroTable[#i] := false;
           // END_IF;
       END_FOR;
   ELSE
       #vibroTable[1] := false;
       #vibroTable[2] := false;
   END_IF;
END_REGION
END_FUNCTION_BLOCK

FUNCTION "preIOtoDB" : Void   // FC3, LAD
{ S7_Optimized_Access := 'TRUE' }
VERSION : 0.1
// stored: AutoNumber true, IsIECCheckEnabled false, SetENOAutomatically false, UDAEnableTagReadback false
   VAR_TEMP
      i : Int;
      j : Int;
      k : Int;
      l : Int;
      "m" : Int;
   END_VAR
BEGIN

REGION Network 1 (SCL): активация катушек для автоматического и ручного режимов
   #i:=0;
   FOR #i := 1 TO 12 DO
       //Bunker_leftOpen
       IF "signalKVSStation".qManualMode.Bunker_leftOpen[#i] OR "signalKVSStation".qAutoMode.Bunker_leftOpen[#i]THEN
           "IO".output.Bunker_leftClose[#i] := true;
           "hmi".weightLine[#i].stateLeftValveWeightPocket := true;
       ELSE
           "IO".output.Bunker_leftClose[#i] := false;
       END_IF;

       //Bunker_leftClose
       IF "signalKVSStation".qManualMode.Bunker_leftClose[#i] OR "signalKVSStation".qAutoMode.Bunker_leftClose[#i] THEN
           "IO".output.Bunker_leftOpen[#i] := TRUE;
           "hmi".weightLine[#i].stateLeftValveWeightPocket := FALSE;
       ELSE
           "IO".output.Bunker_leftOpen[#i] := false;
       END_IF;

       //Bunker_rightOpen
       IF "signalKVSStation".qManualMode.Bunker_rightOpen[#i] OR "signalKVSStation".qAutoMode.Bunker_rightOpen[#i] THEN
           "IO".output.Bunker_rightClose[#i] := true;
           "hmi".weightLine[#i].stateRightValveWeightPocket := true;
       ELSE
           "IO".output.Bunker_rightClose[#i] := false;
       END_IF;

       //Bunker_rightClose
       IF "signalKVSStation".qManualMode.Bunker_rightClose[#i] OR "signalKVSStation".qAutoMode.Bunker_rightClose[#i] THEN
           "IO".output.Bunker_rightOpen[#i] := true;
           "hmi".weightLine[#i].stateRightValveWeightPocket := false;
       ELSE
           "IO".output.Bunker_rightOpen[#i] := false;
       END_IF;

       //Door_open
       IF "signalKVSStation".qManualMode.Door_open[#i] OR "signalKVSStation".qAutoMode.Door_open[#i] THEN
           "IO".output.Door_close[#i] := true;
           "hmi".weightLine[#i].stateValveAfterVibroLot := true;
       ELSE
           "IO".output.Door_close[#i] := false;
       END_IF;

       //Door_close
       IF "signalKVSStation".qManualMode.Door_close[#i] OR "signalKVSStation".qAutoMode.Door_close[#i] THEN
           "IO".output.Door_open[#i] := true;
           "hmi".weightLine[#i].stateValveAfterVibroLot := false;
       ELSE
           "IO".output.Door_open[#i] := false;
       END_IF;

       //vibroLot
       IF "signalKVSStation".qManualMode.vibroLot[#i] OR "signalKVSStation".qAutoMode.vibroLot[#i] THEN
           "IO".output.vibroLot[#i] := true;
           "hmi".weightLine[#i].isVibroLotWork := true;
       ELSE
           "hmi".weightLine[#i].isVibroLotWork := false;
           "IO".output.vibroLot[#i] := false;
       END_IF;

       //теперь все что на два цикла
       IF #i = 1 OR #i = 2 THEN
           //Yq_ReadyDoze
           IF "signalKVSStation".qManualMode.Yq_ReadyDoze[#i] OR "signalKVSStation".qAutoMode.Yq_ReadyDoze[#i] THEN
               "IO".output.Yq_ReadyDoze[#i] := true;
           ELSE
               "IO".output.Yq_ReadyDoze[#i] := false;
           END_IF;

           //Conv_FRV
           IF ("signalKVSStation".qManualMode.Conv_FRV[#i] OR "signalKVSStation".qAutoMode.Conv_FRV[#i]) AND NOT("IO".output.Conv_REV[#i])  THEN
               "IO".output.Conv_FRV[#i] := true;
           ELSE
               "IO".output.Conv_FRV[#i] := false;
           END_IF;

           //Conv_REV
           IF ("signalKVSStation".qManualMode.Conv_REV[#i] OR "signalKVSStation".qAutoMode.Conv_REV[#i]) AND NOT("IO".output.Conv_FRV[#i]) THEN
               "IO".output.Conv_REV[#i] := true;
           ELSE
               "IO".output.Conv_REV[#i] := false;
           END_IF;

           //Обратная связь по работе конвейера
           //
           IF "IO".output.Conv_FRV[#i] OR "IO".output.Conv_REV[#i] THEN
               "hmi".outConvAndPack[#i].isWorkConv := true;
           ELSE
               "hmi".outConvAndPack[#i].isWorkConv := false;
           END_IF;

           //vibroTable
           IF "signalKVSStation".qManualMode.vibroTable[#i] OR "signalKVSStation".qAutoMode.vibroTable[#i] THEN
               "IO".output.vibroTable[#i] := true;
               "hmi".addedVibro.stateVibroTable[#i] := true;
           ELSE
               "IO".output.vibroTable[#i] := false;
               "hmi".addedVibro.stateVibroTable[#i] := false;
           END_IF;


       END_IF;

       //flipper_Up
       IF "signalKVSStation".qManualMode.flipper_Up OR "signalKVSStation".qAutoMode.flipper_Up THEN
           "IO".output.flipper_Down := true;
           "hmi".plavnik.statePlavnik := true;
       ELSE
           "IO".output.flipper_Down := false;
       END_IF;

       //flipper_Down
       IF "signalKVSStation".qManualMode.flipper_Down OR "signalKVSStation".qAutoMode.flipper_Down THEN
           "IO".output.flipper_Up := true;
           "hmi".plavnik.statePlavnik := false;
       ELSE
           "IO".output.flipper_Up := false;
       END_IF;

       //питатель
       IF "signalKVSStation".qManualMode.startInConv OR "signalKVSStation".qAutoMode.startInConv THEN
           "IO".output.convSource := true;
           "hmi".sourceConv.isConvWork := true;
       ELSE
           "IO".output.convSource := false;
           "hmi".sourceConv.isConvWork := false;
       END_IF;

   END_FOR;
END_REGION
END_FUNCTION

FUNCTION "DBtoIO" : Void   // FC2, LAD
{ S7_Optimized_Access := 'TRUE' }
VERSION : 0.1
// stored: AutoNumber true, IsIECCheckEnabled false, SetENOAutomatically false, UDAEnableTagReadback false
BEGIN

REGION Network 1: Конвейер1 - вперед
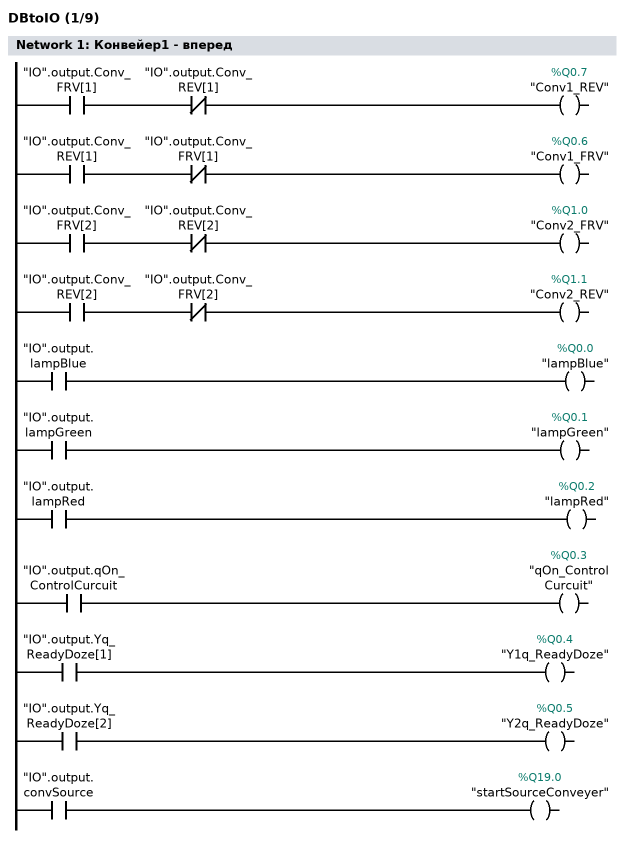
   RUNG wire#powerrail
      Contact( "IO".output.Conv_FRV[1] )
      I_Contact( "IO".output.Conv_REV[1] )
      Coil( "Conv1_REV" )
   END_RUNG
   RUNG wire#powerrail
      Contact( "IO".output.Conv_REV[1] )
      I_Contact( "IO".output.Conv_FRV[1] )
      Coil( "Conv1_FRV" )
   END_RUNG
   RUNG wire#powerrail
      Contact( "IO".output.Conv_FRV[2] )
      I_Contact( "IO".output.Conv_REV[2] )
      Coil( "Conv2_FRV" )
   END_RUNG
   RUNG wire#powerrail
      Contact( "IO".output.Conv_REV[2] )
      I_Contact( "IO".output.Conv_FRV[2] )
      Coil( "Conv2_REV" )
   END_RUNG
   RUNG wire#powerrail
      Contact( "IO".output.lampBlue )
      Coil( "lampBlue" )
   END_RUNG
   RUNG wire#powerrail
      Contact( "IO".output.lampGreen )
      Coil( "lampGreen" )
   END_RUNG
   RUNG wire#powerrail
      Contact( "IO".output.lampRed )
      Coil( "lampRed" )
   END_RUNG
   RUNG wire#powerrail
      Contact( "IO".output.qOn_ControlCurcuit )
      Coil( "qOn_ControlCurcuit" )
   END_RUNG
   RUNG wire#powerrail
      Contact( "IO".output.Yq_ReadyDoze[1] )
      Coil( "Y1q_ReadyDoze" )
   END_RUNG
   RUNG wire#powerrail
      Contact( "IO".output.Yq_ReadyDoze[2] )
      Coil( "Y2q_ReadyDoze" )
   END_RUNG
   RUNG wire#powerrail
      Contact( "IO".output.convSource )
      Coil( "startSourceConveyer" )
   END_RUNG
   // the same network as SCL:
   "Conv1_REV" := "IO".output.Conv_FRV[1] AND NOT "IO".output.Conv_REV[1];
   "Conv1_FRV" := "IO".output.Conv_REV[1] AND NOT "IO".output.Conv_FRV[1];
   "Conv2_FRV" := "IO".output.Conv_FRV[2] AND NOT "IO".output.Conv_REV[2];
   "Conv2_REV" := "IO".output.Conv_REV[2] AND NOT "IO".output.Conv_FRV[2];
   "lampBlue" := "IO".output.lampBlue;
   "lampGreen" := "IO".output.lampGreen;
   "lampRed" := "IO".output.lampRed;
   "qOn_ControlCurcuit" := "IO".output.qOn_ControlCurcuit;
   "Y1q_ReadyDoze" := "IO".output.Yq_ReadyDoze[1];
   "Y2q_ReadyDoze" := "IO".output.Yq_ReadyDoze[2];
   "startSourceConveyer" := "IO".output.convSource;
END_REGION

REGION Network 2: Управление открыванием лопаток - из массива в катушки
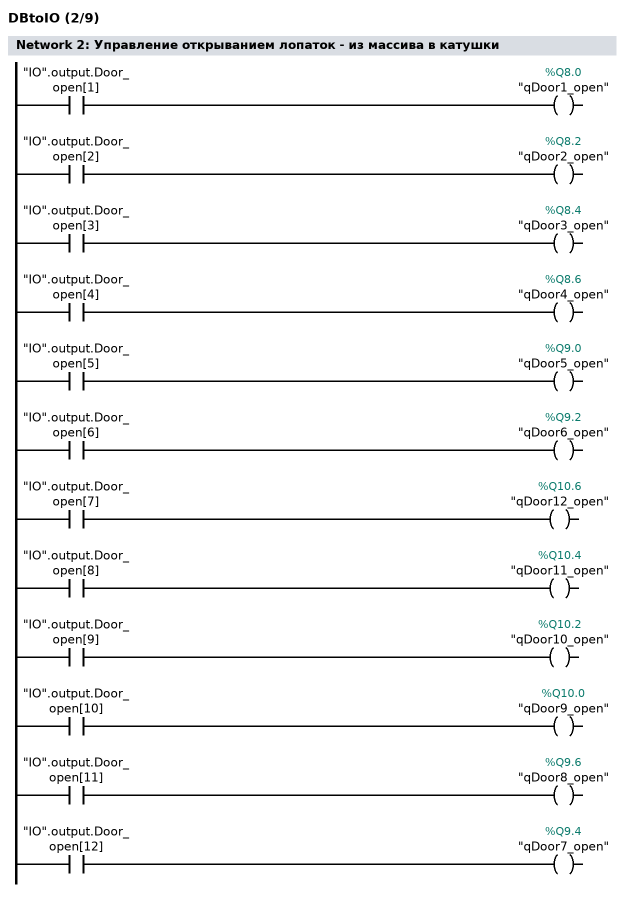
   RUNG wire#powerrail
      Contact( "IO".output.Door_open[1] )
      Coil( "qDoor1_open" )
   END_RUNG
   RUNG wire#powerrail
      Contact( "IO".output.Door_open[2] )
      Coil( "qDoor2_open" )
   END_RUNG
   RUNG wire#powerrail
      Contact( "IO".output.Door_open[3] )
      Coil( "qDoor3_open" )
   END_RUNG
   RUNG wire#powerrail
      Contact( "IO".output.Door_open[4] )
      Coil( "qDoor4_open" )
   END_RUNG
   RUNG wire#powerrail
      Contact( "IO".output.Door_open[5] )
      Coil( "qDoor5_open" )
   END_RUNG
   RUNG wire#powerrail
      Contact( "IO".output.Door_open[6] )
      Coil( "qDoor6_open" )
   END_RUNG
   RUNG wire#powerrail
      Contact( "IO".output.Door_open[7] )
      Coil( "qDoor12_open" )
   END_RUNG
   RUNG wire#powerrail
      Contact( "IO".output.Door_open[8] )
      Coil( "qDoor11_open" )
   END_RUNG
   RUNG wire#powerrail
      Contact( "IO".output.Door_open[9] )
      Coil( "qDoor10_open" )
   END_RUNG
   RUNG wire#powerrail
      Contact( "IO".output.Door_open[10] )
      Coil( "qDoor9_open" )
   END_RUNG
   RUNG wire#powerrail
      Contact( "IO".output.Door_open[11] )
      Coil( "qDoor8_open" )
   END_RUNG
   RUNG wire#powerrail
      Contact( "IO".output.Door_open[12] )
      Coil( "qDoor7_open" )
   END_RUNG
   // the same network as SCL:
   "qDoor1_open" := "IO".output.Door_open[1];
   "qDoor2_open" := "IO".output.Door_open[2];
   "qDoor3_open" := "IO".output.Door_open[3];
   "qDoor4_open" := "IO".output.Door_open[4];
   "qDoor5_open" := "IO".output.Door_open[5];
   "qDoor6_open" := "IO".output.Door_open[6];
   "qDoor12_open" := "IO".output.Door_open[7];
   "qDoor11_open" := "IO".output.Door_open[8];
   "qDoor10_open" := "IO".output.Door_open[9];
   "qDoor9_open" := "IO".output.Door_open[10];
   "qDoor8_open" := "IO".output.Door_open[11];
   "qDoor7_open" := "IO".output.Door_open[12];
END_REGION

REGION Network 3: Управление лопатки закрыть - из массива в катушки
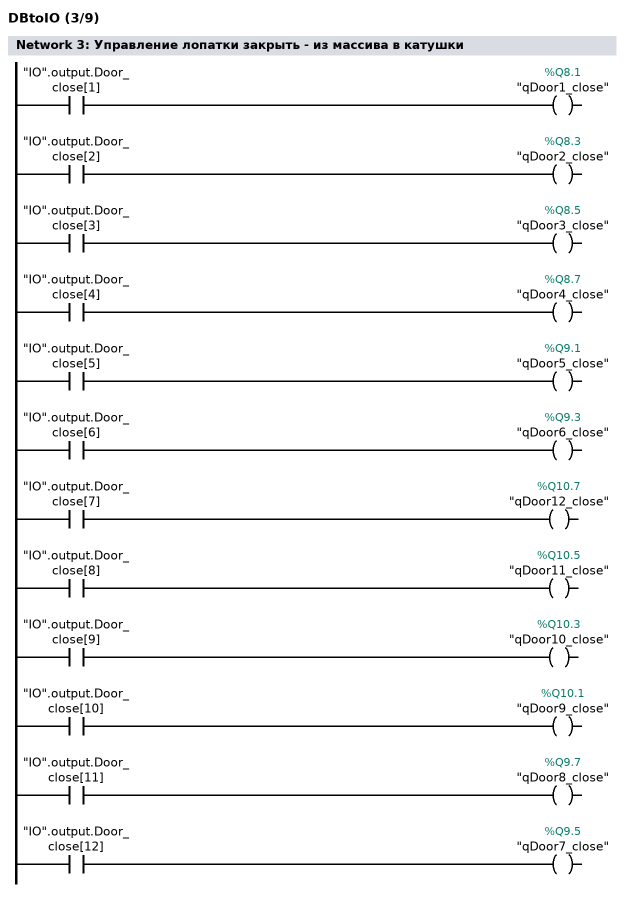
   RUNG wire#powerrail
      Contact( "IO".output.Door_close[1] )
      Coil( "qDoor1_close" )
   END_RUNG
   RUNG wire#powerrail
      Contact( "IO".output.Door_close[2] )
      Coil( "qDoor2_close" )
   END_RUNG
   RUNG wire#powerrail
      Contact( "IO".output.Door_close[3] )
      Coil( "qDoor3_close" )
   END_RUNG
   RUNG wire#powerrail
      Contact( "IO".output.Door_close[4] )
      Coil( "qDoor4_close" )
   END_RUNG
   RUNG wire#powerrail
      Contact( "IO".output.Door_close[5] )
      Coil( "qDoor5_close" )
   END_RUNG
   RUNG wire#powerrail
      Contact( "IO".output.Door_close[6] )
      Coil( "qDoor6_close" )
   END_RUNG
   RUNG wire#powerrail
      Contact( "IO".output.Door_close[7] )
      Coil( "qDoor12_close" )
   END_RUNG
   RUNG wire#powerrail
      Contact( "IO".output.Door_close[8] )
      Coil( "qDoor11_close" )
   END_RUNG
   RUNG wire#powerrail
      Contact( "IO".output.Door_close[9] )
      Coil( "qDoor10_close" )
   END_RUNG
   RUNG wire#powerrail
      Contact( "IO".output.Door_close[10] )
      Coil( "qDoor9_close" )
   END_RUNG
   RUNG wire#powerrail
      Contact( "IO".output.Door_close[11] )
      Coil( "qDoor8_close" )
   END_RUNG
   RUNG wire#powerrail
      Contact( "IO".output.Door_close[12] )
      Coil( "qDoor7_close" )
   END_RUNG
   // the same network as SCL:
   "qDoor1_close" := "IO".output.Door_close[1];
   "qDoor2_close" := "IO".output.Door_close[2];
   "qDoor3_close" := "IO".output.Door_close[3];
   "qDoor4_close" := "IO".output.Door_close[4];
   "qDoor5_close" := "IO".output.Door_close[5];
   "qDoor6_close" := "IO".output.Door_close[6];
   "qDoor12_close" := "IO".output.Door_close[7];
   "qDoor11_close" := "IO".output.Door_close[8];
   "qDoor10_close" := "IO".output.Door_close[9];
   "qDoor9_close" := "IO".output.Door_close[10];
   "qDoor8_close" := "IO".output.Door_close[11];
   "qDoor7_close" := "IO".output.Door_close[12];
END_REGION

REGION Network 4: Управление открыванием левым бункером - из массива в катушки
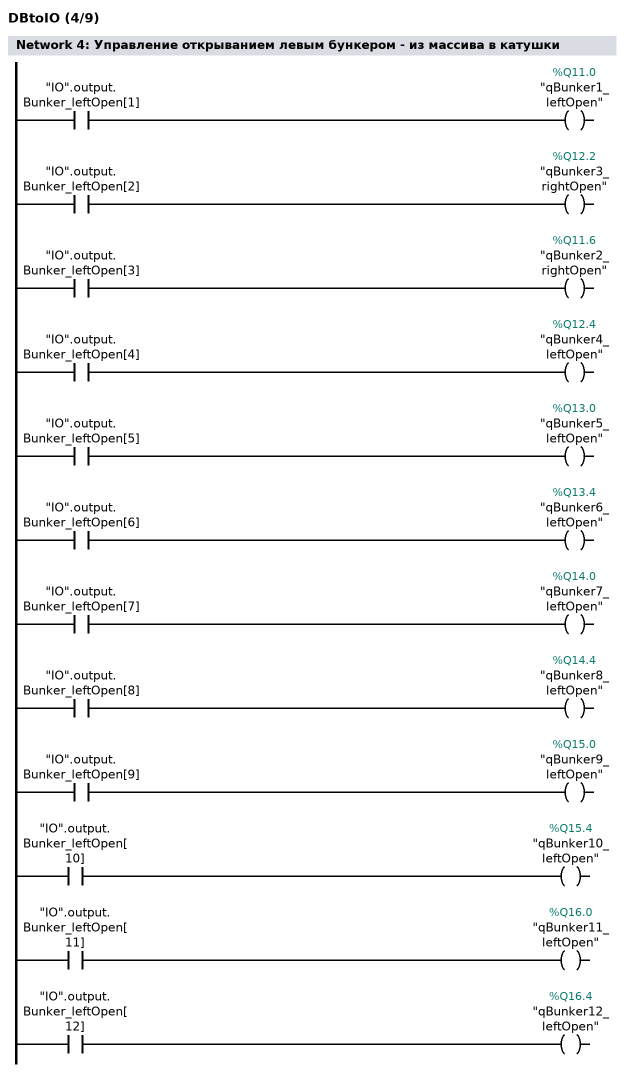
   RUNG wire#powerrail
      Contact( "IO".output.Bunker_leftOpen[1] )
      Coil( "qBunker1_leftOpen" )
   END_RUNG
   RUNG wire#powerrail
      Contact( "IO".output.Bunker_leftOpen[2] )
      Coil( "qBunker3_rightOpen" )
   END_RUNG
   RUNG wire#powerrail
      Contact( "IO".output.Bunker_leftOpen[3] )
      Coil( "qBunker2_rightOpen" )
   END_RUNG
   RUNG wire#powerrail
      Contact( "IO".output.Bunker_leftOpen[4] )
      Coil( "qBunker4_leftOpen" )
   END_RUNG
   RUNG wire#powerrail
      Contact( "IO".output.Bunker_leftOpen[5] )
      Coil( "qBunker5_leftOpen" )
   END_RUNG
   RUNG wire#powerrail
      Contact( "IO".output.Bunker_leftOpen[6] )
      Coil( "qBunker6_leftOpen" )
   END_RUNG
   RUNG wire#powerrail
      Contact( "IO".output.Bunker_leftOpen[7] )
      Coil( "qBunker7_leftOpen" )
   END_RUNG
   RUNG wire#powerrail
      Contact( "IO".output.Bunker_leftOpen[8] )
      Coil( "qBunker8_leftOpen" )
   END_RUNG
   RUNG wire#powerrail
      Contact( "IO".output.Bunker_leftOpen[9] )
      Coil( "qBunker9_leftOpen" )
   END_RUNG
   RUNG wire#powerrail
      Contact( "IO".output.Bunker_leftOpen[10] )
      Coil( "qBunker10_leftOpen" )
   END_RUNG
   RUNG wire#powerrail
      Contact( "IO".output.Bunker_leftOpen[11] )
      Coil( "qBunker11_leftOpen" )
   END_RUNG
   RUNG wire#powerrail
      Contact( "IO".output.Bunker_leftOpen[12] )
      Coil( "qBunker12_leftOpen" )
   END_RUNG
   // the same network as SCL:
   "qBunker1_leftOpen" := "IO".output.Bunker_leftOpen[1];
   "qBunker3_rightOpen" := "IO".output.Bunker_leftOpen[2];
   "qBunker2_rightOpen" := "IO".output.Bunker_leftOpen[3];
   "qBunker4_leftOpen" := "IO".output.Bunker_leftOpen[4];
   "qBunker5_leftOpen" := "IO".output.Bunker_leftOpen[5];
   "qBunker6_leftOpen" := "IO".output.Bunker_leftOpen[6];
   "qBunker7_leftOpen" := "IO".output.Bunker_leftOpen[7];
   "qBunker8_leftOpen" := "IO".output.Bunker_leftOpen[8];
   "qBunker9_leftOpen" := "IO".output.Bunker_leftOpen[9];
   "qBunker10_leftOpen" := "IO".output.Bunker_leftOpen[10];
   "qBunker11_leftOpen" := "IO".output.Bunker_leftOpen[11];
   "qBunker12_leftOpen" := "IO".output.Bunker_leftOpen[12];
END_REGION

REGION Network 5: Управление закрытием левым бункером - из массива в катушки
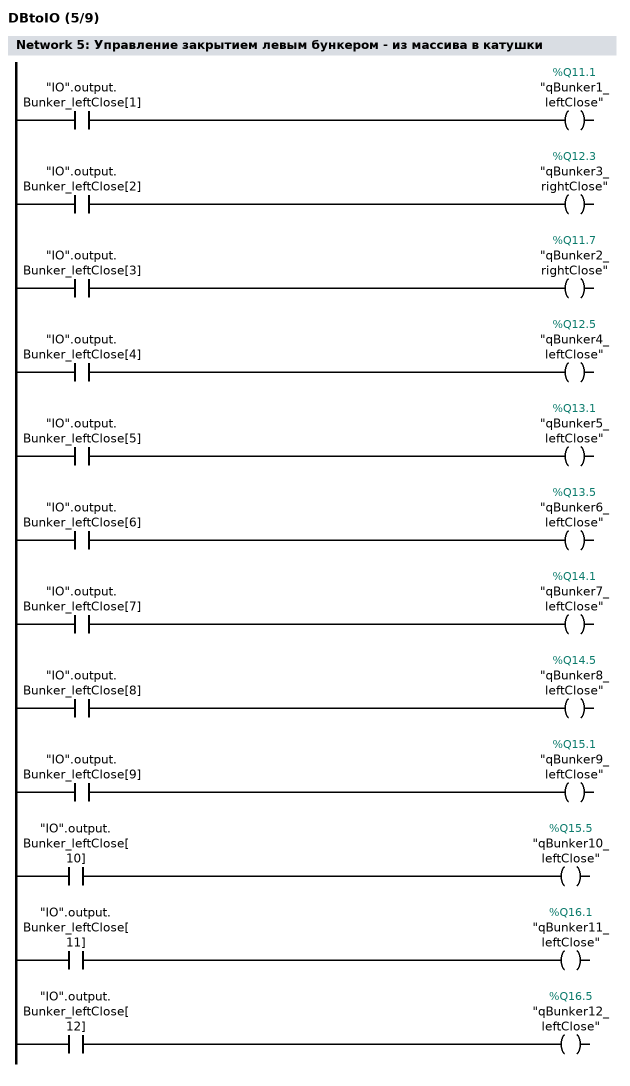
   RUNG wire#powerrail
      Contact( "IO".output.Bunker_leftClose[1] )
      Coil( "qBunker1_leftClose" )
   END_RUNG
   RUNG wire#powerrail
      Contact( "IO".output.Bunker_leftClose[2] )
      Coil( "qBunker3_rightClose" )
   END_RUNG
   RUNG wire#powerrail
      Contact( "IO".output.Bunker_leftClose[3] )
      Coil( "qBunker2_rightClose" )
   END_RUNG
   RUNG wire#powerrail
      Contact( "IO".output.Bunker_leftClose[4] )
      Coil( "qBunker4_leftClose" )
   END_RUNG
   RUNG wire#powerrail
      Contact( "IO".output.Bunker_leftClose[5] )
      Coil( "qBunker5_leftClose" )
   END_RUNG
   RUNG wire#powerrail
      Contact( "IO".output.Bunker_leftClose[6] )
      Coil( "qBunker6_leftClose" )
   END_RUNG
   RUNG wire#powerrail
      Contact( "IO".output.Bunker_leftClose[7] )
      Coil( "qBunker7_leftClose" )
   END_RUNG
   RUNG wire#powerrail
      Contact( "IO".output.Bunker_leftClose[8] )
      Coil( "qBunker8_leftClose" )
   END_RUNG
   RUNG wire#powerrail
      Contact( "IO".output.Bunker_leftClose[9] )
      Coil( "qBunker9_leftClose" )
   END_RUNG
   RUNG wire#powerrail
      Contact( "IO".output.Bunker_leftClose[10] )
      Coil( "qBunker10_leftClose" )
   END_RUNG
   RUNG wire#powerrail
      Contact( "IO".output.Bunker_leftClose[11] )
      Coil( "qBunker11_leftClose" )
   END_RUNG
   RUNG wire#powerrail
      Contact( "IO".output.Bunker_leftClose[12] )
      Coil( "qBunker12_leftClose" )
   END_RUNG
   // the same network as SCL:
   "qBunker1_leftClose" := "IO".output.Bunker_leftClose[1];
   "qBunker3_rightClose" := "IO".output.Bunker_leftClose[2];
   "qBunker2_rightClose" := "IO".output.Bunker_leftClose[3];
   "qBunker4_leftClose" := "IO".output.Bunker_leftClose[4];
   "qBunker5_leftClose" := "IO".output.Bunker_leftClose[5];
   "qBunker6_leftClose" := "IO".output.Bunker_leftClose[6];
   "qBunker7_leftClose" := "IO".output.Bunker_leftClose[7];
   "qBunker8_leftClose" := "IO".output.Bunker_leftClose[8];
   "qBunker9_leftClose" := "IO".output.Bunker_leftClose[9];
   "qBunker10_leftClose" := "IO".output.Bunker_leftClose[10];
   "qBunker11_leftClose" := "IO".output.Bunker_leftClose[11];
   "qBunker12_leftClose" := "IO".output.Bunker_leftClose[12];
END_REGION

REGION Network 6: Управление открыванием правого бункера - из массива в катушки
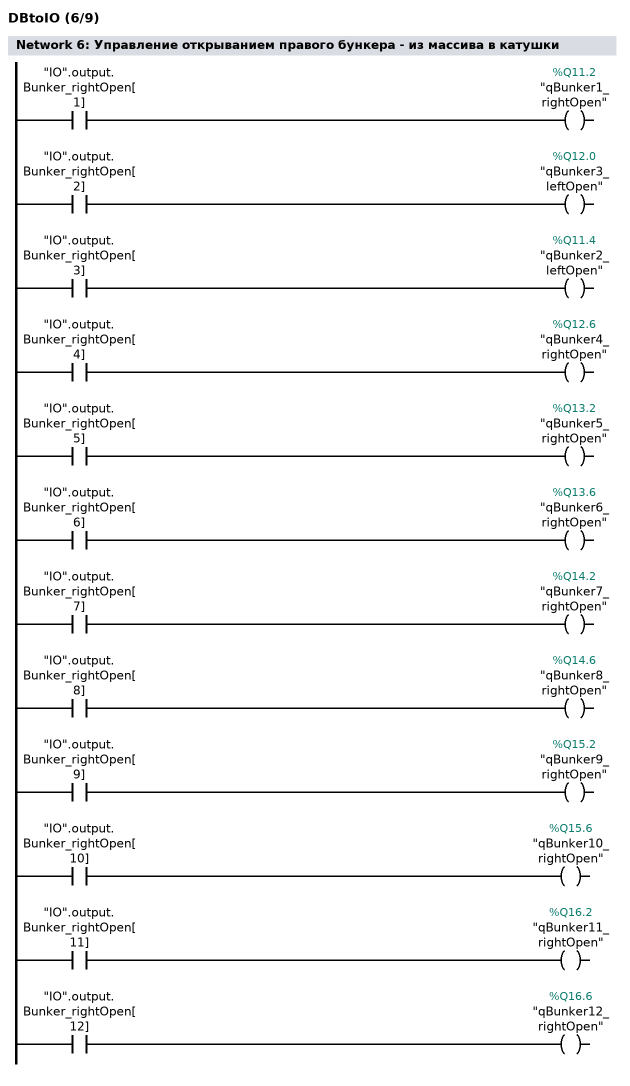
   RUNG wire#powerrail
      Contact( "IO".output.Bunker_rightOpen[1] )
      Coil( "qBunker1_rightOpen" )
   END_RUNG
   RUNG wire#powerrail
      Contact( "IO".output.Bunker_rightOpen[2] )
      Coil( "qBunker3_leftOpen" )
   END_RUNG
   RUNG wire#powerrail
      Contact( "IO".output.Bunker_rightOpen[3] )
      Coil( "qBunker2_leftOpen" )
   END_RUNG
   RUNG wire#powerrail
      Contact( "IO".output.Bunker_rightOpen[4] )
      Coil( "qBunker4_rightOpen" )
   END_RUNG
   RUNG wire#powerrail
      Contact( "IO".output.Bunker_rightOpen[5] )
      Coil( "qBunker5_rightOpen" )
   END_RUNG
   RUNG wire#powerrail
      Contact( "IO".output.Bunker_rightOpen[6] )
      Coil( "qBunker6_rightOpen" )
   END_RUNG
   RUNG wire#powerrail
      Contact( "IO".output.Bunker_rightOpen[7] )
      Coil( "qBunker7_rightOpen" )
   END_RUNG
   RUNG wire#powerrail
      Contact( "IO".output.Bunker_rightOpen[8] )
      Coil( "qBunker8_rightOpen" )
   END_RUNG
   RUNG wire#powerrail
      Contact( "IO".output.Bunker_rightOpen[9] )
      Coil( "qBunker9_rightOpen" )
   END_RUNG
   RUNG wire#powerrail
      Contact( "IO".output.Bunker_rightOpen[10] )
      Coil( "qBunker10_rightOpen" )
   END_RUNG
   RUNG wire#powerrail
      Contact( "IO".output.Bunker_rightOpen[11] )
      Coil( "qBunker11_rightOpen" )
   END_RUNG
   RUNG wire#powerrail
      Contact( "IO".output.Bunker_rightOpen[12] )
      Coil( "qBunker12_rightOpen" )
   END_RUNG
   // the same network as SCL:
   "qBunker1_rightOpen" := "IO".output.Bunker_rightOpen[1];
   "qBunker3_leftOpen" := "IO".output.Bunker_rightOpen[2];
   "qBunker2_leftOpen" := "IO".output.Bunker_rightOpen[3];
   "qBunker4_rightOpen" := "IO".output.Bunker_rightOpen[4];
   "qBunker5_rightOpen" := "IO".output.Bunker_rightOpen[5];
   "qBunker6_rightOpen" := "IO".output.Bunker_rightOpen[6];
   "qBunker7_rightOpen" := "IO".output.Bunker_rightOpen[7];
   "qBunker8_rightOpen" := "IO".output.Bunker_rightOpen[8];
   "qBunker9_rightOpen" := "IO".output.Bunker_rightOpen[9];
   "qBunker10_rightOpen" := "IO".output.Bunker_rightOpen[10];
   "qBunker11_rightOpen" := "IO".output.Bunker_rightOpen[11];
   "qBunker12_rightOpen" := "IO".output.Bunker_rightOpen[12];
END_REGION

REGION Network 7: Управление закрыванием правым бункером - из массива в катушки
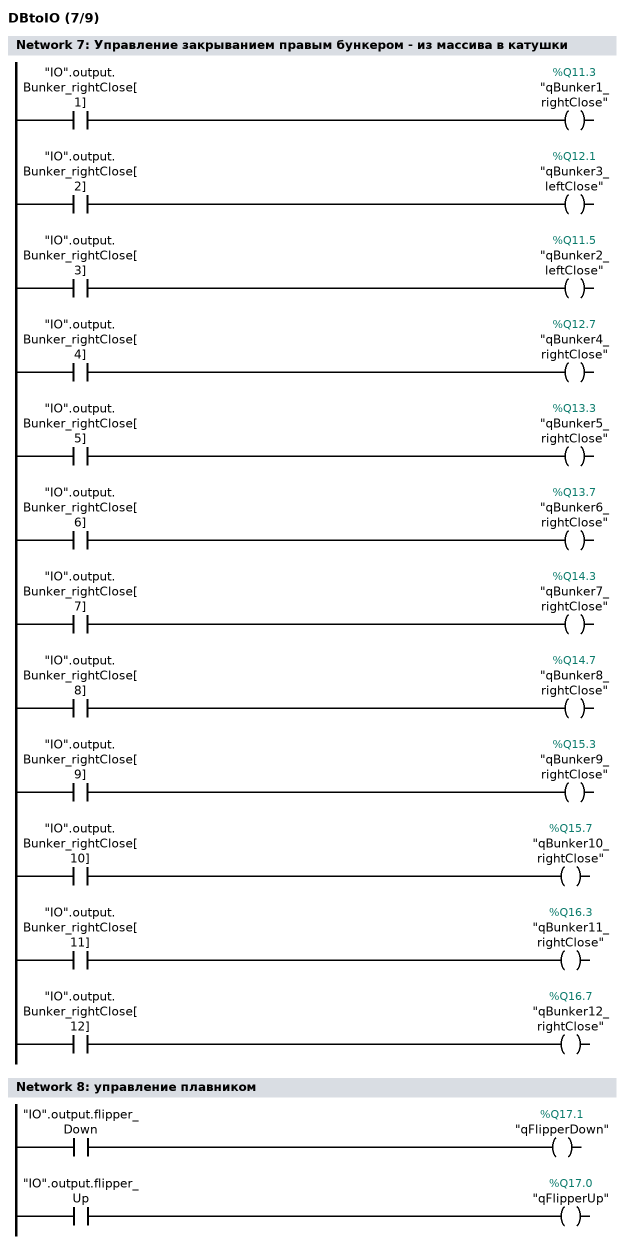
   RUNG wire#powerrail
      Contact( "IO".output.Bunker_rightClose[1] )
      Coil( "qBunker1_rightClose" )
   END_RUNG
   RUNG wire#powerrail
      Contact( "IO".output.Bunker_rightClose[2] )
      Coil( "qBunker3_leftClose" )
   END_RUNG
   RUNG wire#powerrail
      Contact( "IO".output.Bunker_rightClose[3] )
      Coil( "qBunker2_leftClose" )
   END_RUNG
   RUNG wire#powerrail
      Contact( "IO".output.Bunker_rightClose[4] )
      Coil( "qBunker4_rightClose" )
   END_RUNG
   RUNG wire#powerrail
      Contact( "IO".output.Bunker_rightClose[5] )
      Coil( "qBunker5_rightClose" )
   END_RUNG
   RUNG wire#powerrail
      Contact( "IO".output.Bunker_rightClose[6] )
      Coil( "qBunker6_rightClose" )
   END_RUNG
   RUNG wire#powerrail
      Contact( "IO".output.Bunker_rightClose[7] )
      Coil( "qBunker7_rightClose" )
   END_RUNG
   RUNG wire#powerrail
      Contact( "IO".output.Bunker_rightClose[8] )
      Coil( "qBunker8_rightClose" )
   END_RUNG
   RUNG wire#powerrail
      Contact( "IO".output.Bunker_rightClose[9] )
      Coil( "qBunker9_rightClose" )
   END_RUNG
   RUNG wire#powerrail
      Contact( "IO".output.Bunker_rightClose[10] )
      Coil( "qBunker10_rightClose" )
   END_RUNG
   RUNG wire#powerrail
      Contact( "IO".output.Bunker_rightClose[11] )
      Coil( "qBunker11_rightClose" )
   END_RUNG
   RUNG wire#powerrail
      Contact( "IO".output.Bunker_rightClose[12] )
      Coil( "qBunker12_rightClose" )
   END_RUNG
   // the same network as SCL:
   "qBunker1_rightClose" := "IO".output.Bunker_rightClose[1];
   "qBunker3_leftClose" := "IO".output.Bunker_rightClose[2];
   "qBunker2_leftClose" := "IO".output.Bunker_rightClose[3];
   "qBunker4_rightClose" := "IO".output.Bunker_rightClose[4];
   "qBunker5_rightClose" := "IO".output.Bunker_rightClose[5];
   "qBunker6_rightClose" := "IO".output.Bunker_rightClose[6];
   "qBunker7_rightClose" := "IO".output.Bunker_rightClose[7];
   "qBunker8_rightClose" := "IO".output.Bunker_rightClose[8];
   "qBunker9_rightClose" := "IO".output.Bunker_rightClose[9];
   "qBunker10_rightClose" := "IO".output.Bunker_rightClose[10];
   "qBunker11_rightClose" := "IO".output.Bunker_rightClose[11];
   "qBunker12_rightClose" := "IO".output.Bunker_rightClose[12];
END_REGION

REGION Network 8: управление плавником
   RUNG wire#powerrail
      Contact( "IO".output.flipper_Down )
      Coil( "qFlipperDown" )
   END_RUNG
   RUNG wire#powerrail
      Contact( "IO".output.flipper_Up )
      Coil( "qFlipperUp" )
   END_RUNG
   // the same network as SCL:
   "qFlipperDown" := "IO".output.flipper_Down;
   "qFlipperUp" := "IO".output.flipper_Up;
END_REGION

REGION Network 9: Управление вибростолами
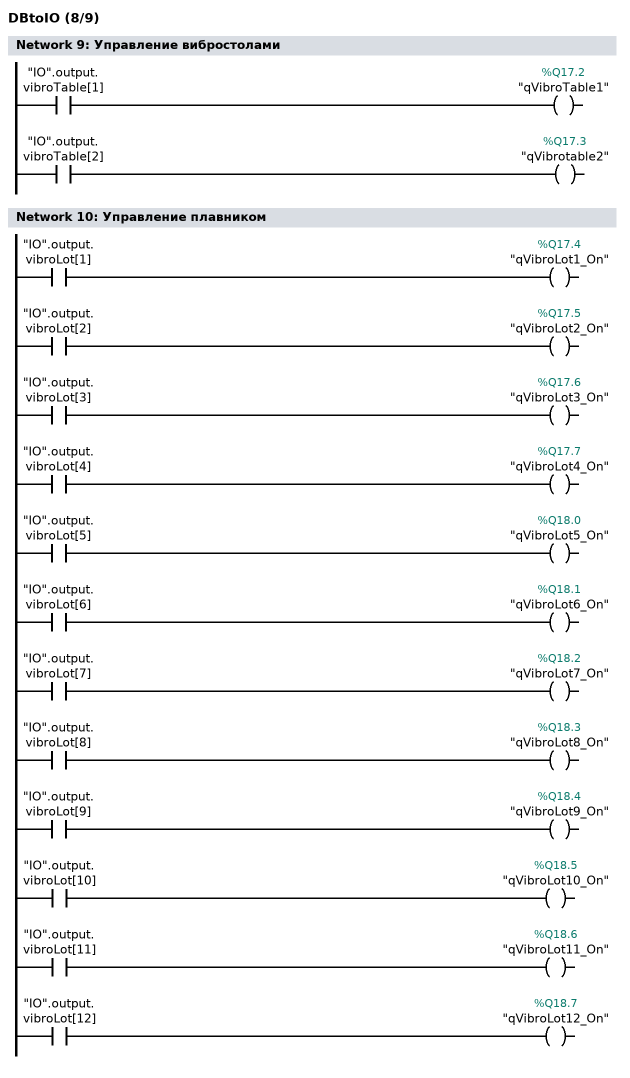
   RUNG wire#powerrail
      Contact( "IO".output.vibroTable[1] )
      Coil( "qVibroTable1" )
   END_RUNG
   RUNG wire#powerrail
      Contact( "IO".output.vibroTable[2] )
      Coil( "qVibrotable2" )
   END_RUNG
   // the same network as SCL:
   "qVibroTable1" := "IO".output.vibroTable[1];
   "qVibrotable2" := "IO".output.vibroTable[2];
END_REGION

REGION Network 10: Управление плавником
   RUNG wire#powerrail
      Contact( "IO".output.vibroLot[1] )
      Coil( "qVibroLot1_On" )
   END_RUNG
   RUNG wire#powerrail
      Contact( "IO".output.vibroLot[2] )
      Coil( "qVibroLot2_On" )
   END_RUNG
   RUNG wire#powerrail
      Contact( "IO".output.vibroLot[3] )
      Coil( "qVibroLot3_On" )
   END_RUNG
   RUNG wire#powerrail
      Contact( "IO".output.vibroLot[4] )
      Coil( "qVibroLot4_On" )
   END_RUNG
   RUNG wire#powerrail
      Contact( "IO".output.vibroLot[5] )
      Coil( "qVibroLot5_On" )
   END_RUNG
   RUNG wire#powerrail
      Contact( "IO".output.vibroLot[6] )
      Coil( "qVibroLot6_On" )
   END_RUNG
   RUNG wire#powerrail
      Contact( "IO".output.vibroLot[7] )
      Coil( "qVibroLot7_On" )
   END_RUNG
   RUNG wire#powerrail
      Contact( "IO".output.vibroLot[8] )
      Coil( "qVibroLot8_On" )
   END_RUNG
   RUNG wire#powerrail
      Contact( "IO".output.vibroLot[9] )
      Coil( "qVibroLot9_On" )
   END_RUNG
   RUNG wire#powerrail
      Contact( "IO".output.vibroLot[10] )
      Coil( "qVibroLot10_On" )
   END_RUNG
   RUNG wire#powerrail
      Contact( "IO".output.vibroLot[11] )
      Coil( "qVibroLot11_On" )
   END_RUNG
   RUNG wire#powerrail
      Contact( "IO".output.vibroLot[12] )
      Coil( "qVibroLot12_On" )
   END_RUNG
   // the same network as SCL:
   "qVibroLot1_On" := "IO".output.vibroLot[1];
   "qVibroLot2_On" := "IO".output.vibroLot[2];
   "qVibroLot3_On" := "IO".output.vibroLot[3];
   "qVibroLot4_On" := "IO".output.vibroLot[4];
   "qVibroLot5_On" := "IO".output.vibroLot[5];
   "qVibroLot6_On" := "IO".output.vibroLot[6];
   "qVibroLot7_On" := "IO".output.vibroLot[7];
   "qVibroLot8_On" := "IO".output.vibroLot[8];
   "qVibroLot9_On" := "IO".output.vibroLot[9];
   "qVibroLot10_On" := "IO".output.vibroLot[10];
   "qVibroLot11_On" := "IO".output.vibroLot[11];
   "qVibroLot12_On" := "IO".output.vibroLot[12];
END_REGION

REGION Network 11: Задание уставки вибрации
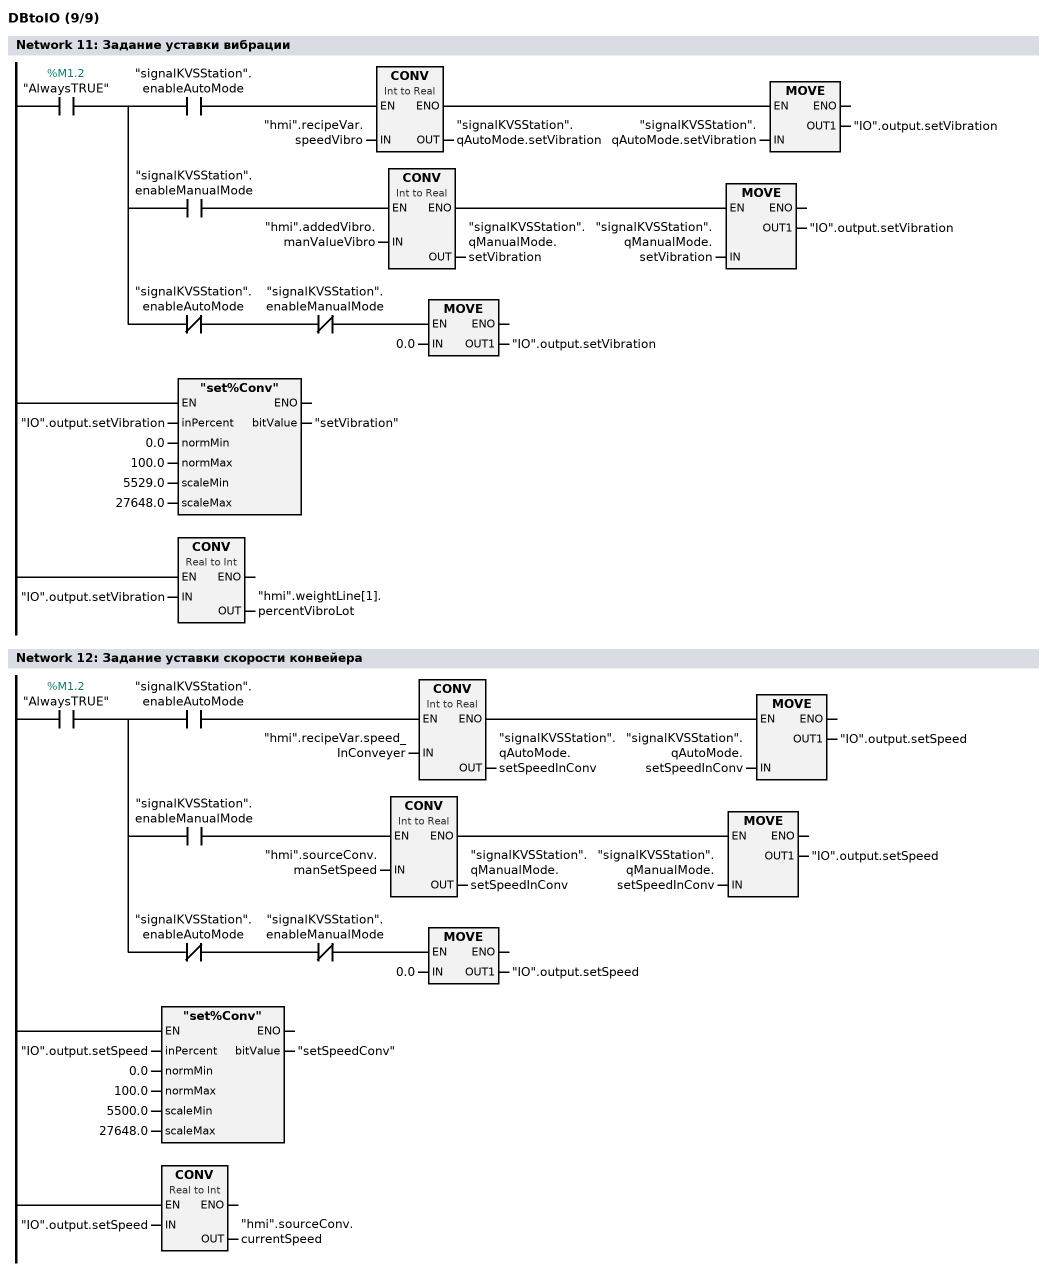
   RUNG wire#powerrail
      Contact( "AlwaysTRUE" )
      wire#w1
      Contact( "signalKVSStation".enableAutoMode )
      { S7_Templates := "[SrcType := Int, DestType := Real]" } Convert(in := "hmi".recipeVar.speedVibro, out => "signalKVSStation".qAutoMode.setVibration)
      Move(in := "signalKVSStation".qAutoMode.setVibration, out1 => "IO".output.setVibration)
   END_RUNG
   RUNG wire#w1
      Contact( "signalKVSStation".enableManualMode )
      { S7_Templates := "[SrcType := Int, DestType := Real]" } Convert(in := "hmi".addedVibro.manValueVibro, out => "signalKVSStation".qManualMode.setVibration)
      Move(in := "signalKVSStation".qManualMode.setVibration, out1 => "IO".output.setVibration)
   END_RUNG
   RUNG wire#w1
      I_Contact( "signalKVSStation".enableAutoMode )
      I_Contact( "signalKVSStation".enableManualMode )
      Move(in := 0.0, out1 => "IO".output.setVibration)
   END_RUNG
   RUNG wire#powerrail
      "set%Conv"(inPercent := "IO".output.setVibration, normMin := 0.0, normMax := 100.0, scaleMin := 5529.0, scaleMax := 27648.0, bitValue => "setVibration")
   END_RUNG
   RUNG wire#powerrail
      { S7_Templates := "[SrcType := Real, DestType := Int]" } Convert(in := "IO".output.setVibration, out => "hmi".weightLine[1].percentVibroLot)
   END_RUNG
   // the same network as SCL:
   IF "AlwaysTRUE" AND "signalKVSStation".enableAutoMode THEN
       "signalKVSStation".qAutoMode.setVibration := INT_TO_REAL("hmi".recipeVar.speedVibro);
       "IO".output.setVibration := "signalKVSStation".qAutoMode.setVibration;
   END_IF;
   IF "AlwaysTRUE" AND "signalKVSStation".enableManualMode THEN
       "signalKVSStation".qManualMode.setVibration := INT_TO_REAL("hmi".addedVibro.manValueVibro);
       "IO".output.setVibration := "signalKVSStation".qManualMode.setVibration;
   END_IF;
   IF "AlwaysTRUE" AND NOT "signalKVSStation".enableAutoMode AND NOT "signalKVSStation".enableManualMode THEN
       "IO".output.setVibration := 0.0;
   END_IF;
   "set%Conv"(inPercent := "IO".output.setVibration,
              normMin := 0.0,
              normMax := 100.0,
              scaleMin := 5529.0,
              scaleMax := 27648.0,
              bitValue => "setVibration");
   "hmi".weightLine[1].percentVibroLot := REAL_TO_INT("IO".output.setVibration);
END_REGION

REGION Network 12: Задание уставки скорости конвейера
   RUNG wire#powerrail
      Contact( "AlwaysTRUE" )
      wire#w1
      Contact( "signalKVSStation".enableAutoMode )
      { S7_Templates := "[SrcType := Int, DestType := Real]" } Convert(in := "hmi".recipeVar.speed_InConveyer, out => "signalKVSStation".qAutoMode.setSpeedInConv)
      Move(in := "signalKVSStation".qAutoMode.setSpeedInConv, out1 => "IO".output.setSpeed)
   END_RUNG
   RUNG wire#w1
      Contact( "signalKVSStation".enableManualMode )
      { S7_Templates := "[SrcType := Int, DestType := Real]" } Convert(in := "hmi".sourceConv.manSetSpeed, out => "signalKVSStation".qManualMode.setSpeedInConv)
      Move(in := "signalKVSStation".qManualMode.setSpeedInConv, out1 => "IO".output.setSpeed)
   END_RUNG
   RUNG wire#w1
      I_Contact( "signalKVSStation".enableAutoMode )
      I_Contact( "signalKVSStation".enableManualMode )
      Move(in := 0.0, out1 => "IO".output.setSpeed)
   END_RUNG
   RUNG wire#powerrail
      "set%Conv"(inPercent := "IO".output.setSpeed, normMin := 0.0, normMax := 100.0, scaleMin := 5500.0, scaleMax := 27648.0, bitValue => "setSpeedConv")
   END_RUNG
   RUNG wire#powerrail
      { S7_Templates := "[SrcType := Real, DestType := Int]" } Convert(in := "IO".output.setSpeed, out => "hmi".sourceConv.currentSpeed)
   END_RUNG
   // the same network as SCL:
   IF "AlwaysTRUE" AND "signalKVSStation".enableAutoMode THEN
       "signalKVSStation".qAutoMode.setSpeedInConv := INT_TO_REAL("hmi".recipeVar.speed_InConveyer);
       "IO".output.setSpeed := "signalKVSStation".qAutoMode.setSpeedInConv;
   END_IF;
   IF "AlwaysTRUE" AND "signalKVSStation".enableManualMode THEN
       "signalKVSStation".qManualMode.setSpeedInConv := INT_TO_REAL("hmi".sourceConv.manSetSpeed);
       "IO".output.setSpeed := "signalKVSStation".qManualMode.setSpeedInConv;
   END_IF;
   IF "AlwaysTRUE" AND NOT "signalKVSStation".enableAutoMode AND NOT "signalKVSStation".enableManualMode THEN
       "IO".output.setSpeed := 0.0;
   END_IF;
   "set%Conv"(inPercent := "IO".output.setSpeed,
              normMin := 0.0,
              normMax := 100.0,
              scaleMin := 5500.0,
              scaleMax := 27648.0,
              bitValue => "setSpeedConv");
   "hmi".sourceConv.currentSpeed := REAL_TO_INT("IO".output.setSpeed);
END_REGION
END_FUNCTION

FUNCTION "set%Conv" : Void   // FC4, LAD
{ S7_Optimized_Access := 'TRUE' }
VERSION : 0.1
// stored: AutoNumber true, IsIECCheckEnabled false, SetENOAutomatically false, UDAEnableTagReadback false
   VAR_INPUT
      inPercent : Real;
      normMin : Real;
      normMax : Real;
      scaleMin : Real;
      scaleMax : Real;
   END_VAR
   VAR_OUTPUT
      bitValue : Int;
   END_VAR
   VAR_TEMP
      temp : Real;
   END_VAR
BEGIN

REGION Network 1
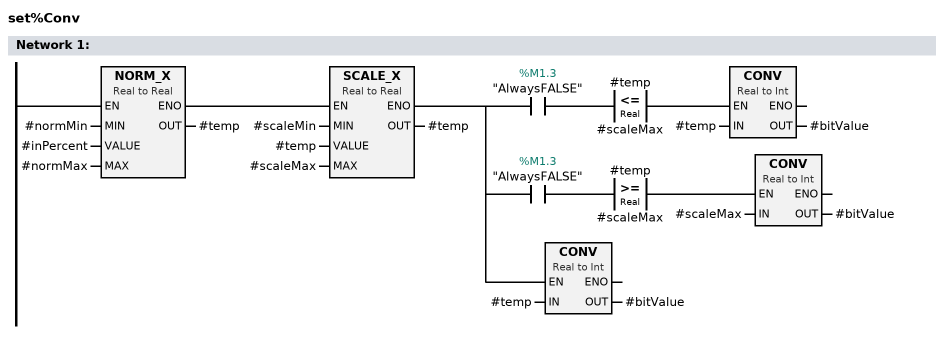
   RUNG wire#powerrail
      { S7_Templates := "[SrcType := Real, DestType := Real]" } Normalize(min := #normMin, value := #inPercent, max := #normMax, out => #temp)
      { S7_Templates := "[SrcType := Real, DestType := Real]" } Scale(min := #scaleMin, value := #temp, max := #scaleMax, out => #temp)
      wire#w1
      Contact( "AlwaysFALSE" )
      { S7_Templates := "SrcType := Real" } LE_Contact(in1 := #temp, in2 := #scaleMax)
      { S7_Templates := "[SrcType := Real, DestType := Int]" } Convert(in := #temp, out => #bitValue)
   END_RUNG
   RUNG wire#w1
      Contact( "AlwaysFALSE" )
      { S7_Templates := "SrcType := Real" } GE_Contact(in1 := #temp, in2 := #scaleMax)
      { S7_Templates := "[SrcType := Real, DestType := Int]" } Convert(in := #scaleMax, out => #bitValue)
   END_RUNG
   RUNG wire#w1
      { S7_Templates := "[SrcType := Real, DestType := Int]" } Convert(in := #temp, out => #bitValue)
   END_RUNG
   // the same network as SCL:
   #temp := NORM_X(MIN := #normMin, VALUE := #inPercent, MAX := #normMax);
   #temp := SCALE_X(MIN := #scaleMin, VALUE := #temp, MAX := #scaleMax);
   IF "AlwaysFALSE" AND (#temp <= #scaleMax) THEN #bitValue := REAL_TO_INT(#temp); END_IF;
   IF "AlwaysFALSE" AND (#temp >= #scaleMax) THEN #bitValue := REAL_TO_INT(#scaleMax); END_IF;
   #bitValue := REAL_TO_INT(#temp);
END_REGION
END_FUNCTION

FUNCTION "alarmBlock" : Void   // FC10, LAD
{ S7_Optimized_Access := 'TRUE' }
VERSION : 0.1
// stored: AutoNumber true, IsIECCheckEnabled false, SetENOAutomatically false, UDAEnableTagReadback false
   VAR_TEMP
      i : DInt;
   END_VAR
BEGIN

REGION Network 1: Тепловое реле Конв1
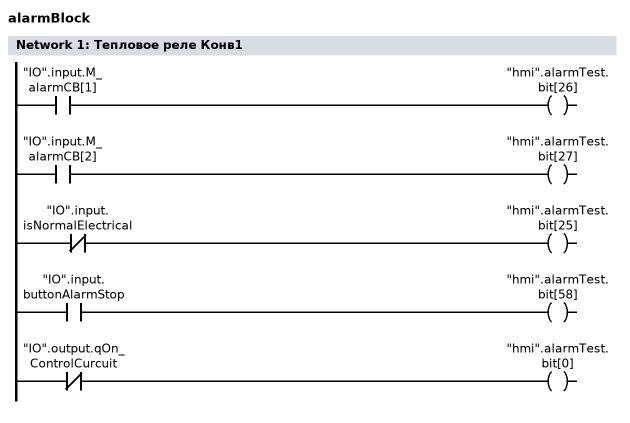
   RUNG wire#powerrail
      Contact( "IO".input.M_alarmCB[1] )
      Coil( "hmi".alarmTest.bit[26] )
   END_RUNG
   RUNG wire#powerrail
      Contact( "IO".input.M_alarmCB[2] )
      Coil( "hmi".alarmTest.bit[27] )
   END_RUNG
   RUNG wire#powerrail
      I_Contact( "IO".input.isNormalElectrical )
      Coil( "hmi".alarmTest.bit[25] )
   END_RUNG
   RUNG wire#powerrail
      Contact( "IO".input.buttonAlarmStop )
      Coil( "hmi".alarmTest.bit[58] )
   END_RUNG
   RUNG wire#powerrail
      I_Contact( "IO".output.qOn_ControlCurcuit )
      Coil( "hmi".alarmTest.bit[0] )
   END_RUNG
   // the same network as SCL:
   "hmi".alarmTest.bit[26] := "IO".input.M_alarmCB[1];
   "hmi".alarmTest.bit[27] := "IO".input.M_alarmCB[2];
   "hmi".alarmTest.bit[25] := NOT "IO".input.isNormalElectrical;
   "hmi".alarmTest.bit[58] := "IO".input.buttonAlarmStop;
   "hmi".alarmTest.bit[0] := NOT "IO".output.qOn_ControlCurcuit;
END_REGION

REGION Network 2 (SCL): обрывы весовых датчиков
   #i := 0;
   FOR #i := 1 TO 12 DO
       IF "signalKVSStation".currentWeight[#i] > 7000 THEN
           "hmi".alarmTest.bit[12 + #i] := true;
       ELSE
           "hmi".alarmTest.bit[12 + #i] := false;
       END_IF;
   END_FOR;
END_REGION

REGION Network 3 (SCL)
   #i := 0;
   FOR #i := 0 TO 70 DO
       IF "hmi".alarmTest.bit[#i] THEN
           "hmi".commonAlarm := true;
           EXIT;
       END_IF;
       IF #i = 70 THEN
           "hmi".commonAlarm := false;
       END_IF;
   END_FOR;
END_REGION
END_FUNCTION

ORGANIZATION_BLOCK "Time error interrupt"   // OB80, LAD, TimeErrorInterrupt
{ S7_Optimized_Access := 'TRUE' }
VERSION : 0.1
// stored: IsIECCheckEnabled false, SetENOAutomatically false
   VAR_INPUT
      Fault_ID : Byte;   // Fault identifier
      Csg_OBnr : OB_ANY;   // Number of OB causing the error
      Csg_Prio : UInt;   // Priority of OB causing the error
   END_VAR
BEGIN
END_ORGANIZATION_BLOCK

FUNCTION "bitMaskSortFor" : Void   // FC6, LAD
{ S7_Optimized_Access := 'TRUE' }
VERSION : 0.1
// stored: AutoNumber true, IsIECCheckEnabled false, SetENOAutomatically false, UDAEnableTagReadback false
   VAR_INPUT
      value : DInt;
   END_VAR
   VAR_IN_OUT
      bitMask : Array[0..12] of Bool;
   END_VAR
BEGIN

REGION Network 1 (SCL)
   #bitMask[0] := #value.%X0;
   #bitMask[1] := #value.%X1;
   #bitMask[2] := #value.%X2;
   #bitMask[3] := #value.%X3;
   #bitMask[4] := #value.%X4;
   #bitMask[5] := #value.%X5;
   #bitMask[6] := #value.%X6;
   #bitMask[7] := #value.%X7;
   #bitMask[8] := #value.%X8;
   #bitMask[9] := #value.%X9;
   #bitMask[10] := #value.%X10;
   #bitMask[11] := #value.%X11;
   #bitMask[12] := #value.%X12;
END_REGION
END_FUNCTION

FUNCTION "findSum" : Void   // FC8, LAD
{ S7_Optimized_Access := 'TRUE' }
VERSION : 0.1
// stored: AutoNumber true, IsIECCheckEnabled false, SetENOAutomatically false, UDAEnableTagReadback false
   VAR_INPUT
      arrWeight : Array[0..12] of Real;
      arrBitMask : Array[0..12] of Bool;
   END_VAR
   VAR_IN_OUT
      tmpSum : Real;
   END_VAR
BEGIN

REGION Network 1 (SCL)
   #tmpSum := #arrWeight[0] * BOOL_TO_INT(#arrBitMask[0]) +
   #arrWeight[1] * BOOL_TO_INT(#arrBitMask[1])+
   #arrWeight[2] * BOOL_TO_INT(#arrBitMask[2]) +
   #arrWeight[3] * BOOL_TO_INT(#arrBitMask[3]) +
   #arrWeight[4] * BOOL_TO_INT(#arrBitMask[4]) +
   #arrWeight[5] * BOOL_TO_INT(#arrBitMask[5]) +
   #arrWeight[6] * BOOL_TO_INT(#arrBitMask[6]) +
   #arrWeight[7] * BOOL_TO_INT(#arrBitMask[7]) +
   #arrWeight[8] * BOOL_TO_INT(#arrBitMask[8]) +
   #arrWeight[9] * BOOL_TO_INT(#arrBitMask[9]) +
   #arrWeight[10] * BOOL_TO_INT(#arrBitMask[10]) +
   #arrWeight[11] * BOOL_TO_INT(#arrBitMask[11]) +
   #arrWeight[12] * BOOL_TO_INT(#arrBitMask[12]);
END_REGION
END_FUNCTION

FUNCTION "pushToArray" : Void   // FC5, LAD
{ S7_Optimized_Access := 'TRUE' }
VERSION : 0.1
// stored: AutoNumber true, IsIECCheckEnabled false, SetENOAutomatically false, UDAEnableTagReadback false
   VAR_INPUT
      addValue : Real;
   END_VAR
   VAR_IN_OUT
      "array" : Array[*] of Real;
   END_VAR
   VAR_TEMP
      lowIndex : DInt;
      highIndex : DInt;
      i : SInt;
   END_VAR
BEGIN

REGION Network 1 (SCL)
   #lowIndex := LOWER_BOUND(ARR := #array, DIM := 1);
   #highIndex := UPPER_BOUND(ARR := #array, DIM := 1);

   #i := 0;
   FOR #i := (#highIndex - 1) TO #lowIndex BY -1 DO 
       #array[#i+1] := #array[#i];
   END_FOR;
   #array[#lowIndex] := #addValue;

   ENO := true;
END_REGION
END_FUNCTION

FUNCTION_BLOCK "tst"
{ S7_Optimized_Access := 'TRUE' }
VERSION : 0.1
   VAR 
      abcDec : DInt;
      arrBin : Array[1..12] of Bool;
      qwer : Array[0..12] of Real := [0.0, 5.0, 1.1, 2.2, 6.5, 3.3, 4.4, 5.5, 6.9, 7.7, 8.8, 9.9, 10.2];
      Sort_Real_Instance : "Sort_Real";
   END_VAR

   VAR_TEMP 
      i : SInt;
   END_VAR


BEGIN
	REGION
	    
	        #arrBin[1] := #abcDec.%X0;
	        #arrBin[2] := #abcDec.%X1;
	        #arrBin[3] := #abcDec.%X2;
	        #arrBin[4] := #abcDec.%X3;
	        #arrBin[5] := #abcDec.%X4;
	        #arrBin[6] := #abcDec.%X5;
	        #arrBin[7] := #abcDec.%X6;
	        #arrBin[8] := #abcDec.%X7;
	        #arrBin[9] := #abcDec.%X8;
	        #arrBin[10] := #abcDec.%X9;
	        #arrBin[11] := #abcDec.%X10;
	        #arrBin[12] := #abcDec.%X11;
	        
	    END_REGION ;
	    #Sort_Real_Instance(sortDirection:=true,
	                        array:=#qwer);
	    
	    
END_FUNCTION_BLOCK

FUNCTION "rcvDataWeight" : Void
{ S7_Optimized_Access := 'TRUE' }
VERSION : 0.1
   VAR_INPUT 
      ADDR_DEVICE : UInt;
      Ton_changeStep : Bool;
   END_VAR

   VAR_IN_OUT 
      Ton_Start : Bool;
      Step : SInt;
      MB_MASTER : Struct
         REQ : Bool;
         MB_ADDR : UInt;
         MODE : USInt;
         DATA_ADDR : UDInt;
         DATA_LEN : UInt;
         DONE : Bool;
         BUSY : Bool;
         ERROR : Bool;
      END_STRUCT;
   END_VAR


BEGIN
	        #Ton_Start := TRUE;
	        
	        #MB_MASTER.MB_ADDR := #ADDR_DEVICE;
	        #MB_MASTER.MODE := 0;
	        #MB_MASTER.DATA_ADDR := 40064;
	        #MB_MASTER.DATA_LEN := 2;
	        #MB_MASTER.REQ := TRUE;
	        
	        IF NOT (#MB_MASTER.BUSY) AND
	            (#MB_MASTER.DONE OR
	            #Ton_changeStep OR #MB_MASTER.ERROR) THEN
	            #MB_MASTER.REQ  := FALSE;
	            #Ton_Start := FALSE;
	            #Step := #Step + 1;
	        END_IF;
END_FUNCTION

FUNCTION "sndCALIBR&Tara" : Void
{ S7_Optimized_Access := 'TRUE' }
VERSION : 0.1
   VAR_INPUT 
      ADDR_DEVICE : UInt;   // адрес опрашиваемого устройства
      ton_changeStep : Bool;   // таймер на переход следующего шага опроса
   END_VAR

   VAR_IN_OUT 
      MB_MASTER : Struct
         REQ : Bool;
         MB_ADDR : UInt;
         MODE : USInt;
         DATA_ADDR : UDInt;
         DATA_LEN : UInt;
         DONE : Bool;
         BUSY : Bool;
         ERROR : Bool;
      END_STRUCT;
      Ton_Start : Bool;   // сигнал на старт таймера
      Buffer : Array[0..20] of Word;   // буффер данных у блока мастера модбаса
      Step : SInt;   // текущий шаг
      Calibrate : Bool;   // сигнал на калибровку
      Tara : Bool;   // сигнал на тарирование
   END_VAR


BEGIN
	        IF #Calibrate OR//калибровка
	            #Tara//тарирование
	        THEN
	            #Ton_Start := TRUE;
	            
	            #MB_MASTER.MB_ADDR := #ADDR_DEVICE;
	            #MB_MASTER.MODE := 1;
	            #MB_MASTER.DATA_ADDR := 40068;
	            #MB_MASTER.DATA_LEN := 1;
	            #MB_MASTER.REQ := TRUE;
	            
	            IF #Calibrate THEN
	                #Buffer[0] := 16#C2FA;
	            ELSIF #Tara THEN
	                #Buffer[0] := 16#C1BA;
	            END_IF;
	            
	            IF NOT (#MB_MASTER.BUSY) AND
	                (#MB_MASTER.DONE OR
	                #ton_changeStep OR
	                #MB_MASTER.ERROR) THEN
	                #MB_MASTER.REQ := FALSE;
	                #Ton_Start := FALSE;
	                #Step := #Step + 1;
	                IF #Calibrate THEN
	                    #Calibrate := FALSE;
	                ELSIF #Tara THEN
	                    #Tara := false;
	                END_IF;
	                    
	                #Buffer[0] := 0;
	            END_IF;
	        ELSE
	            #Step := #Step + 1;
	            #MB_MASTER.REQ := FALSE;
	        END_IF;
	        
	       
	            
END_FUNCTION

FUNCTION "sndVibration" : Void
{ S7_Optimized_Access := 'TRUE' }
VERSION : 0.1
   VAR_INPUT 
      ADDR_DEVICE : UInt;   // адрес опрашиваемого устройства
      ton_changeStep : Bool;   // таймер на переход следующего шага опроса
   END_VAR

   VAR_IN_OUT 
      MB_MASTER : Struct
         REQ : Bool;
         MB_ADDR : UInt;
         MODE : USInt;
         DATA_ADDR : UDInt;
         DATA_LEN : UInt;
         DONE : Bool;
         BUSY : Bool;
         ERROR : Bool;
      END_STRUCT;
      Ton_Start : Bool;   // сигнал на старт таймера
      Buffer : Array[0..20] of Word;   // буффер данных у блока мастера модбаса
      Step : SInt;   // текущий шаг
   END_VAR

   VAR_TEMP 
      i : SInt;
   END_VAR


BEGIN
	            #Ton_Start := TRUE;
	            
	            #MB_MASTER.MB_ADDR := #ADDR_DEVICE;
	            #MB_MASTER.MODE := 1;
	            #MB_MASTER.DATA_ADDR := 40001;
	            #MB_MASTER.DATA_LEN := 8;
	            #MB_MASTER.REQ := TRUE;
	            
	            #i := 0;
	            FOR #i := 0 TO 7 DO
	                #Buffer[#i] := INT_TO_WORD(REAL_TO_INT("IO".output.setVibration * 10.0));
	            END_FOR;
	            IF "signalKVSStation".enableAutoMode THEN
	                #Buffer[2] := INT_TO_WORD(1000);
	            END_IF;
	            
	            IF NOT(#MB_MASTER.BUSY) AND
	                (#MB_MASTER.DONE OR
	                #ton_changeStep OR
	                #MB_MASTER.ERROR) THEN
	                #MB_MASTER.REQ := FALSE;
	                #Ton_Start := FALSE;
	                #Step := #Step + 1;
	                #Buffer[0] := 0;
	            END_IF;
	        
	        
	       
	            
END_FUNCTION

DATA_BLOCK "AutoMode_DB"   // DB5
VERSION : 0.1
// stored: AutoNumber true, DBAccessibleFromOPCUA true, InstanceOfName AutoMode, InstanceOfType FB
"AutoMode"
BEGIN
END_DATA_BLOCK

DATA_BLOCK "ManualMode_DB"   // DB30
VERSION : 0.1
// stored: AutoNumber false, DBAccessibleFromOPCUA true, InstanceOfName ManualMode, InstanceOfType FB
"ManualMode"
BEGIN
END_DATA_BLOCK

DATA_BLOCK "tst_DB"   // DB6
VERSION : 0.1
// stored: AutoNumber true, DBAccessibleFromOPCUA true, InstanceOfName tst, InstanceOfType FB
"tst"
BEGIN
END_DATA_BLOCK

DATA_BLOCK "modbus_FB_DB"   // DB3
VERSION : 0.1
// stored: AutoNumber true, DBAccessibleFromOPCUA true, InstanceOfName modbus_FB, InstanceOfType FB
"modbus_FB"
BEGIN
END_DATA_BLOCK

DATA_BLOCK "IEC_Counter_0_DB"   // DB7
{ S7_Optimized_Access := 'TRUE' }
// stored: AutoNumber true, DBAccessibleFromOPCUA true, InstanceOfName IEC_COUNTER, OfSystemLibElement IEC_COUNTER, OfSystemLibVersion 1.0
"IEC_COUNTER"
   // VAR RETAIN
   //    CU : Bool;
   //    CD : Bool;
   //    R : Bool;
   //    LD : Bool;
   //    QU : Bool;
   //    QD : Bool;
   //    PV : Int;
   //    CV : Int;
   // END_VAR
BEGIN
END_DATA_BLOCK

DATA_BLOCK "IEC_Timer_TEST"   // DB8
{ S7_Optimized_Access := 'TRUE' }
// stored: AutoNumber true, DBAccessibleFromOPCUA true, InstanceOfName IEC_TIMER, OfSystemLibElement IEC_TIMER, OfSystemLibVersion 1.0
"IEC_TIMER"
   // VAR
   //    PT : Time;
   //    ET { ExternalWritable := 'False'} : Time;
   //    IN : Bool;
   //    Q { ExternalWritable := 'False'} : Bool;
   // END_VAR
BEGIN
END_DATA_BLOCK

DATA_BLOCK "IEC_Timer_TEST_HIGH"   // DB9
{ S7_Optimized_Access := 'TRUE' }
// stored: AutoNumber true, DBAccessibleFromOPCUA true, InstanceOfName IEC_TIMER, OfSystemLibElement IEC_TIMER, OfSystemLibVersion 1.0
"IEC_TIMER"
   // VAR
   //    PT : Time;
   //    ET { ExternalWritable := 'False'} : Time;
   //    IN : Bool;
   //    Q { ExternalWritable := 'False'} : Bool;
   // END_VAR
BEGIN
END_DATA_BLOCK

DATA_BLOCK "isWorkAM"   // DB2
{ S7_Optimized_Access := 'TRUE' }
// stored: AutoNumber true, DBAccessibleFromOPCUA true, InstanceOfName IEC_TIMER, OfSystemLibElement IEC_TIMER, OfSystemLibVersion 1.0
"IEC_TIMER"
   // VAR
   //    PT : Time;
   //    ET { ExternalWritable := 'False'} : Time;
   //    IN : Bool;
   //    Q { ExternalWritable := 'False'} : Bool;
   // END_VAR
BEGIN
END_DATA_BLOCK

DATA_BLOCK "onControlCircuit"   // DB1
{ S7_Optimized_Access := 'TRUE' }
// stored: AutoNumber true, DBAccessibleFromOPCUA true, InstanceOfName IEC_TIMER, OfSystemLibElement IEC_TIMER, OfSystemLibVersion 1.0
"IEC_TIMER"
   // VAR
   //    PT : Time;
   //    ET { ExternalWritable := 'False'} : Time;
   //    IN : Bool;
   //    Q { ExternalWritable := 'False'} : Bool;
   // END_VAR
BEGIN
END_DATA_BLOCK
